// TIA Portal project "Sorting Plant Control" (V16)

(* hardware
DEVICE "S71500/ET200MP station_1"  S7-1500 station
   slot 0: "Rail_0"  Rack  6ES7 590-1***0-0AA0
   slot 0: "PM 190W 120/230VAC"  PM 190W 120/230VAC  6EP1333-4BA00
   slot 1: "Sorting Plant Controller"  CPU 1516F-3 PN/DP  6ES7 516-3FN02-0AB0  V2.8
      slot 3: "CPU display_1"  6ES7591-1BA00-0AA0
      slot 32768: "PROFINET interface_1"  X1
         slot 32769: "Port_1"  X1 P1
         slot 32770: "Port_2"  X1 P2
      slot 33024: "PROFINET interface_2"  X2
         slot 33025: "Port_1"  X2 P1
      slot 33280: "DP interface_1"  X3
      slot 34817: "Virtual CP interface port_1"  Virtual CP interface port  Virtual CP interface port
   slot 2: "DI 32x24VDC HF_1"  DI 32x24VDC HF  6ES7 521-1BL00-0AB0  V2.2
   slot 3: "DQ 32x24VDC/0.5A HF_1"  DQ 32x24VDC/0.5A HF  6ES7 522-1BL01-0AB0  V1.1
   slot 4: "AI 8xU/I/RTD/TC ST_1"  AI 8xU/I/RTD/TC ST  6ES7 531-7KF00-0AB0  V2.2
   slot 5: "AQ 4xU/I ST_1"  AQ 4xU/I ST  6ES7 532-5HD00-0AB0  V2.2
DEVICE "HMI"  TP900 Comfort
   slot 0: "HMI"  TP900 Comfort  6AV2 124-0JC01-0AX0  16.0.0.0
   slot 1: "HMI_RT_5"  TP900 Comfort  6AV2 124-0JC01-0AX0  16.0.0.0
   slot 5: "HMI._CP_1"  PROFINET Interface  16.0.0.0
      slot 1: "PROFINET Interface_1"  PROFINET Interface
         slot 1: "Port_1"  Port
         slot 2: "Port_2"  Port
   slot 7: "HMI.I/DP_CP_1"  MPI/DP Interface  16.0.0.0
*)

// ===== PLC "Sorting Plant Controller"  CPU 1516F-3 PN/DP =====

VAR_GLOBAL   // PLC tag table "Default tag table"
   "System_Byte" AT %MB1 : Byte;
   "FirstScan" AT %M1.0 : Bool;
   "DiagStatusUpdate" AT %M1.1 : Bool;
   "AlwaysTRUE" AT %M1.2 : Bool;
   "AlwaysFALSE" AT %M1.3 : Bool;
   "Clock_Byte" AT %MB0 : Byte;
   "Clock_10Hz" AT %M0.0 : Bool;
   "Clock_5Hz" AT %M0.1 : Bool;
   "Clock_2.5Hz" AT %M0.2 : Bool;
   "Clock_2Hz" AT %M0.3 : Bool;
   "Clock_1.25Hz" AT %M0.4 : Bool;
   "Clock_1Hz" AT %M0.5 : Bool;
   "Clock_0.625Hz" AT %M0.6 : Bool;
   "Clock_0.5Hz" AT %M0.7 : Bool;
   "Tag_1" AT %M2.0 : Bool;
   "Tag_2" AT %M2.1 : Bool;
   "Tag_3" AT %M2.2 : Bool;
   "Tag_4" AT %M2.3 : Bool;
   "Tag_5" AT %M2.4 : Bool;
   "Tag_6" AT %M2.5 : Bool;
   "Tag_7" AT %M2.6 : Bool;
   "Tag_8" AT %M2.7 : Bool;
END_VAR

VAR_GLOBAL   // PLC tag table "Sorting Plant Tags"
   "csLightSensorCube_Detected" AT %I0.0 : Bool;   // 0: cube workpiece not detected; 1: cube workpiece detected by the light sensor
   "csLightSensorCylinder_Detected" AT %I0.1 : Bool;   // 0: cylinder workpiece not detected; 1: cylinder workpiece detected by the light sensor
   "csLightSensorWorkpiece_Detected" AT %I0.2 : Bool;   // 0: light sensor did not detect a workpiece, 1: light sensor detected a workpiece
   "csLimitSwitchCylinderNotExtended_Activated" AT %I0.3 : Bool;   // 0: the cylinder is fully extended; 1: the cylinder is not fully extended
   "csLimitSwitchCylinderRetracted_Activated" AT %I0.4 : Bool;   // 0: the cylinder is not fully retracted; 1: the cylinder is fully retracted
   "osWorkpieceCylinder_SetActive" AT %Q0.0 : Bool;   // 0: cylinder workpiece are not produced; 1: cylinder workpiece are produced
   "osWorkpieceCube_SetActive" AT %Q0.1 : Bool;   // 0: cube workpiece are not produced; 1: cube workpiece are produced
   "pcCylinderHeadRetract_SetActive" AT %Q0.2 : Bool;   // 0: do not retract push cylinder; 1: retract push cylinder
   "pcCylinderHeadExtend_SetActive" AT %Q0.3 : Bool;   // 0: do not extend push cylinder; 1: extend push cylinder
   "scConveyorLongConstSpeed_SetActive" AT %Q0.4 : Bool;   // 0: do not move the long conveyor at constant speed; 1: move the long conveyor at constant speed
   "scConveyorLongVarSpeed_SetActive" AT %Q0.5 : Bool;   // 0: do not move the long conveyor at variable speed; 1: move the long conveyor at variable speed
   "scConveyorShortConstSpeed_SetActive" AT %Q0.6 : Bool;   // 0: do not move the short conveyor at constant speed; 1: move the short conveyor at constant speed
   "scConveyorShortVarSpeed_SetActive" AT %Q0.7 : Bool;   // 0: do not move the short conveyor at variable speed; 1: move the short conveyor at variable speed
   "scConveyorLongVarSpeed_SetSpeed" AT %QD64 : Real;   // variable velocity for long conveyor belt in m/s
   "scConveyorShortVarSpeed_SetSpeed" AT %QD68 : Real;   // variable velocity for short conveyor belt in m/s
END_VAR

DATA_BLOCK "Control_HMI"   // DB1
{ S7_Optimized_Access := 'TRUE' }
VERSION : 0.1
   VAR RETAIN
      toHMI : Struct
         resetStatus : Bool;
         numWorkpieces : USInt;
         numCylinders : USInt;
         numCubes : USInt;
         Error : Bool;
         ErrorID : Word;
      END_STRUCT;
      fromHMI : Struct
         resetSimulation : Bool;
         generateWorkpieces : Bool;
         cylinderCommand : Struct
            extendCylinder : Bool;
            retractCylinder : Bool;
         END_STRUCT;
         shortConveyor : Struct
            constSpeedControl : Bool;
            varSpeedControl : Bool;
            varSpeedPercentage : Real;   // % value
         END_STRUCT;
         longConveyor : Struct
            constSpeedControl : Bool;
            varSpeedControl : Bool;
            varSpeedPercentage : Real;   // % value
         END_STRUCT;
      END_STRUCT;
   END_VAR
BEGIN
END_DATA_BLOCK

DATA_BLOCK "SortingPlantControl_DB"   // DB2
{ S7_Optimized_Access := 'TRUE' }
VERSION : 0.1
// stored: InstanceOfName SortingPlantControl
"SortingPlantControl"
BEGIN
END_DATA_BLOCK

FUNCTION_BLOCK "SortingPlantControl"   // FB1, LAD
{ S7_Optimized_Access := 'TRUE' }
VERSION : 0.1
   VAR_INPUT
      "Light Sensor Cube" : Bool;
      "Light Sensor Cylinder" : Bool;
      "Light Sensor Workpiece" : Bool;
      "Limit Switch Cylinder NotExtended" : Bool;
      "Limit Switch Cylinder Retracted" : Bool;
      "Cylinder Extend Command" : Bool;
      "Cylinder Retract Command" : Bool;
      "Long Conveyor Constant Speed Command" : Bool;
      "Long Conveyor Var Speed Command" : Bool;
      "Long Conveyor Var Speed Percentage" : Real;
      "Short Conveyor Constant Speed Command" : Bool;
      "Short Conveyor Var Speed Command" : Bool;
      "Short Conveyor Var Speed Percentage" : Real;
      "Generate Workpieces" : Bool;
      "Total Workpiece Counter Value" : USInt;
      "Cylinder Counter Value" : USInt;
      "Cube Counter Value" : USInt;
   END_VAR
   VAR_OUTPUT
      Error : Bool;
      ErrorID : Word;
      "Workpiece Cylinder Generation" : Bool;
      "Workpiece Cube Generation" : Bool;
      "Cylinder Retract" : Bool;
      "Cylinder Extend" : Bool;
      "Conveyor Long Const Speed" : Bool;
      "Conveyor Long Var Speed" : Bool;
      "Conveyor Long Var Speed Setpoint" : Real;
      "Conveyor Short Const Speed" : Bool;
      "Conveyor Short Var Speed" : Bool;
      "Conveyor Long Short Speed Setpoint" : Real;
      "Total Workpiece Count Set" : USInt;
      "Cylinder Count Set" : USInt;
      "Cube Count Set" : USInt;
   END_VAR
   VAR
      CylinderControl_Instance : "CylinderControl";
      ShortConveyorControl_Instance : "ConveyorControl";
      LongConveyorControl_Instance : "ConveyorControl";
      upCounter_Workpiece : CTU_USINT;
      lightSensorWorkpieceFALLEdge : Bool;
      lightSensorCubeFALLEdge : Bool;
      upCounter_Cube : CTU_USINT;
      lightSensorCylinderFALLEdge : Bool;
      upCounter_Cylinder : CTU_USINT;
      waitTime : Time;   // in ms
      startWaitTimer : Bool;
      onTimer_Waitfunction : TON_TIME;
      cylinderInterlock : Bool;
      shortConvInterlock : Bool;
      longConvInterlock : Bool;
   END_VAR
   VAR_TEMP
      shortConvFault : Bool;
      longConvFault : Bool;
      cylFault : Bool;
      waitTimeCalc : UDInt;
      performEject : Bool;
   END_VAR
   VAR CONSTANT
      constantMaxSpeed : Real := 0.05;   // max speed in m/s for constant speed mode
      varMaxSpeed : Real := 0.15;   // max speed in m/s for variable speed mode
      optimumEjectDistance : Real := 0.02;   // optimal distance for ejection in m. In this case 20 mm
   END_VAR
   VAR_TEMP   // added for the SCL form of the ladder/FBD networks
      _w1 : Bool;
      _w2 : Bool;
      _w3 : Bool;
   END_VAR
BEGIN

REGION Network 1: Generate workpieces when triggered from HMI
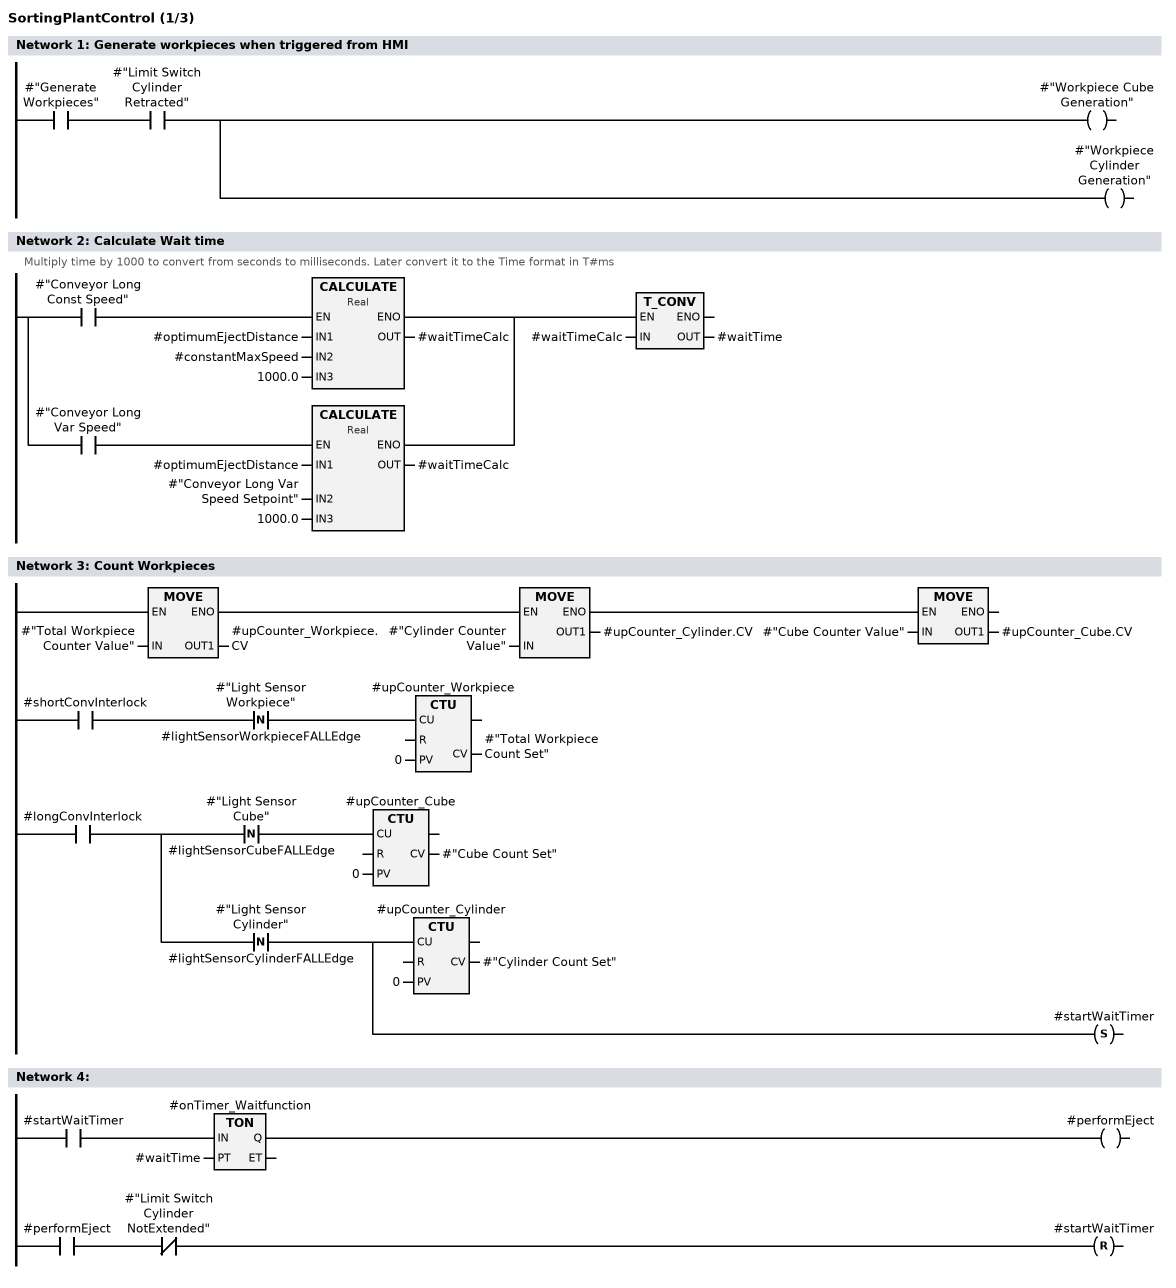
   RUNG wire#powerrail
      Contact( #"Generate Workpieces" )
      Contact( #"Limit Switch Cylinder Retracted" )
      wire#w1
      Coil( #"Workpiece Cube Generation" )
   END_RUNG
   RUNG wire#w1
      Coil( #"Workpiece Cylinder Generation" )
   END_RUNG
   // the same network as SCL:
   #"Workpiece Cube Generation" := #"Generate Workpieces" AND #"Limit Switch Cylinder Retracted";
   #"Workpiece Cylinder Generation" := #"Workpiece Cube Generation";
END_REGION

REGION Network 2: Calculate Wait time
   // Multiply time by 1000 to convert from seconds to milliseconds. Later convert it to the Time format in T#ms
   IF #"Conveyor Long Const Speed" THEN
       #waitTimeCalc := (#optimumEjectDistance / #constantMaxSpeed) * 1000.0;
   END_IF;
   IF #"Conveyor Long Var Speed" THEN
       #waitTimeCalc := (#optimumEjectDistance / #"Conveyor Long Var Speed Setpoint") * 1000.0;
   END_IF;
   IF #"Conveyor Long Const Speed" OR #"Conveyor Long Var Speed" THEN
       #waitTime := T_CONV(IN := #waitTimeCalc);
   END_IF;
END_REGION

REGION Network 3: Count Workpieces
   #upCounter_Workpiece.CV := #"Total Workpiece Counter Value";
   #upCounter_Cylinder.CV := #"Cylinder Counter Value";
   #upCounter_Cube.CV := #"Cube Counter Value";
   #_w1 := #shortConvInterlock AND NOT #"Light Sensor Workpiece" AND #lightSensorWorkpieceFALLEdge;   // falling edge of #"Light Sensor Workpiece"
   #lightSensorWorkpieceFALLEdge := #"Light Sensor Workpiece";
   #upCounter_Workpiece(CU := #_w1, PV := 0, CV => #"Total Workpiece Count Set");   // CTU
   #_w2 := #longConvInterlock AND NOT #"Light Sensor Cube" AND #lightSensorCubeFALLEdge;   // falling edge of #"Light Sensor Cube"
   #lightSensorCubeFALLEdge := #"Light Sensor Cube";
   #upCounter_Cube(CU := #_w2, PV := 0, CV => #"Cube Count Set");   // CTU
   #_w3 := #longConvInterlock AND NOT #"Light Sensor Cylinder" AND #lightSensorCylinderFALLEdge;   // falling edge of #"Light Sensor Cylinder"
   #lightSensorCylinderFALLEdge := #"Light Sensor Cylinder";
   #upCounter_Cylinder(CU := #_w3, PV := 0, CV => #"Cylinder Count Set");   // CTU
   IF #_w3 THEN #startWaitTimer := TRUE; END_IF;
END_REGION

REGION Network 4
   #onTimer_Waitfunction(IN := #startWaitTimer, PT := #waitTime);   // TON
   #performEject := #onTimer_Waitfunction.Q;
   IF #performEject AND NOT #"Limit Switch Cylinder NotExtended" THEN #startWaitTimer := FALSE; END_IF;
END_REGION

REGION Network 5: Control Pneumatic Cylinder
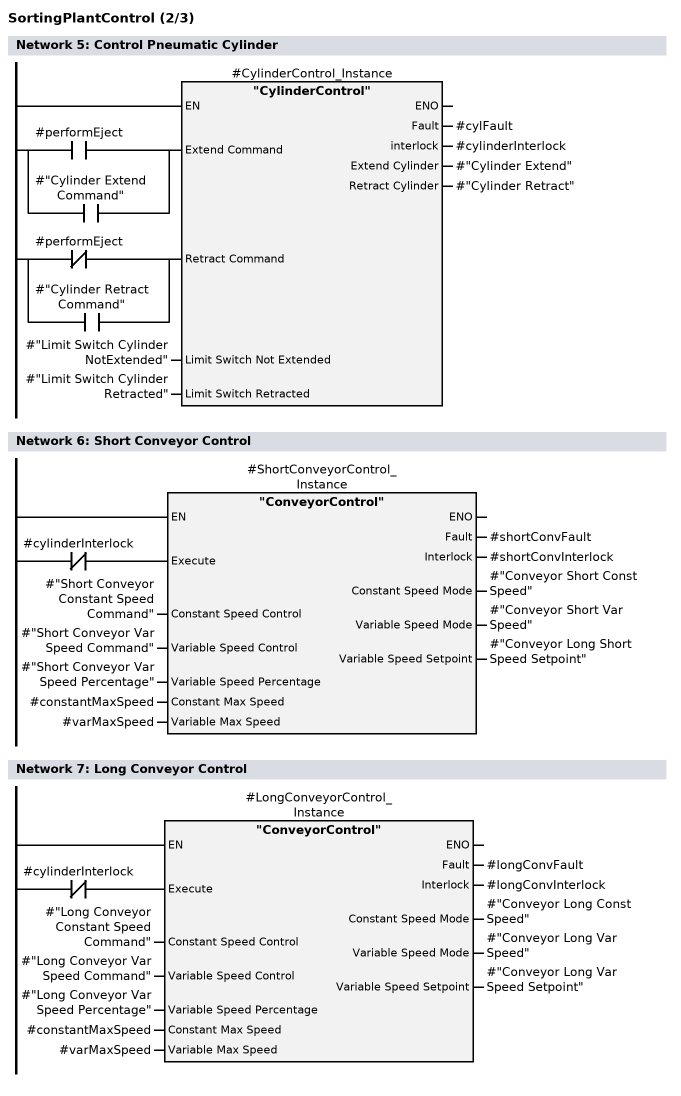
   RUNG wire#powerrail
      #CylinderControl_Instance("Extend Command" := wire#w1, "Retract Command" := wire#w2, "Limit Switch Not Extended" := #"Limit Switch Cylinder NotExtended", "Limit Switch Retracted" := #"Limit Switch Cylinder Retracted", Fault => #cylFault, interlock => #cylinderInterlock, "Extend Cylinder" => #"Cylinder Extend", "Retract Cylinder" => #"Cylinder Retract")
   END_RUNG
   RUNG wire#powerrail
      Contact( #performEject )
   END_RUNG wire#w1
   RUNG wire#powerrail
      Contact( #"Cylinder Extend Command" )
   END_RUNG wire#w1
   RUNG wire#powerrail
      I_Contact( #performEject )
   END_RUNG wire#w2
   RUNG wire#powerrail
      Contact( #"Cylinder Retract Command" )
   END_RUNG wire#w2
   // the same network as SCL:
   #CylinderControl_Instance("Extend Command" := #performEject OR #"Cylinder Extend Command",   // "CylinderControl"
                           "Retract Command" := NOT #performEject OR #"Cylinder Retract Command",
                           "Limit Switch Not Extended" := #"Limit Switch Cylinder NotExtended",
                           "Limit Switch Retracted" := #"Limit Switch Cylinder Retracted",
                           Fault => #cylFault,
                           interlock => #cylinderInterlock,
                           "Extend Cylinder" => #"Cylinder Extend",
                           "Retract Cylinder" => #"Cylinder Retract");
END_REGION

REGION Network 6: Short Conveyor Control
   RUNG wire#powerrail
      #ShortConveyorControl_Instance(Execute := wire#w1, "Constant Speed Control" := #"Short Conveyor Constant Speed Command", "Variable Speed Control" := #"Short Conveyor Var Speed Command", "Variable Speed Percentage" := #"Short Conveyor Var Speed Percentage", "Constant Max Speed" := #constantMaxSpeed, "Variable Max Speed" := #varMaxSpeed, Fault => #shortConvFault, Interlock => #shortConvInterlock, "Constant Speed Mode" => #"Conveyor Short Const Speed", "Variable Speed Mode" => #"Conveyor Short Var Speed", "Variable Speed Setpoint" => #"Conveyor Long Short Speed Setpoint")
   END_RUNG
   RUNG wire#powerrail
      I_Contact( #cylinderInterlock )
   END_RUNG wire#w1
   // the same network as SCL:
   #ShortConveyorControl_Instance(Execute := NOT #cylinderInterlock,   // "ConveyorControl"
                           "Constant Speed Control" := #"Short Conveyor Constant Speed Command",
                           "Variable Speed Control" := #"Short Conveyor Var Speed Command",
                           "Variable Speed Percentage" := #"Short Conveyor Var Speed Percentage",
                           "Constant Max Speed" := #constantMaxSpeed,
                           "Variable Max Speed" := #varMaxSpeed,
                           Fault => #shortConvFault,
                           Interlock => #shortConvInterlock,
                           "Constant Speed Mode" => #"Conveyor Short Const Speed",
                           "Variable Speed Mode" => #"Conveyor Short Var Speed",
                           "Variable Speed Setpoint" => #"Conveyor Long Short Speed Setpoint");
END_REGION

REGION Network 7: Long Conveyor Control
   RUNG wire#powerrail
      #LongConveyorControl_Instance(Execute := wire#w1, "Constant Speed Control" := #"Long Conveyor Constant Speed Command", "Variable Speed Control" := #"Long Conveyor Var Speed Command", "Variable Speed Percentage" := #"Long Conveyor Var Speed Percentage", "Constant Max Speed" := #constantMaxSpeed, "Variable Max Speed" := #varMaxSpeed, Fault => #longConvFault, Interlock => #longConvInterlock, "Constant Speed Mode" => #"Conveyor Long Const Speed", "Variable Speed Mode" => #"Conveyor Long Var Speed", "Variable Speed Setpoint" => #"Conveyor Long Var Speed Setpoint")
   END_RUNG
   RUNG wire#powerrail
      I_Contact( #cylinderInterlock )
   END_RUNG wire#w1
   // the same network as SCL:
   #LongConveyorControl_Instance(Execute := NOT #cylinderInterlock,   // "ConveyorControl"
                           "Constant Speed Control" := #"Long Conveyor Constant Speed Command",
                           "Variable Speed Control" := #"Long Conveyor Var Speed Command",
                           "Variable Speed Percentage" := #"Long Conveyor Var Speed Percentage",
                           "Constant Max Speed" := #constantMaxSpeed,
                           "Variable Max Speed" := #varMaxSpeed,
                           Fault => #longConvFault,
                           Interlock => #longConvInterlock,
                           "Constant Speed Mode" => #"Conveyor Long Const Speed",
                           "Variable Speed Mode" => #"Conveyor Long Var Speed",
                           "Variable Speed Setpoint" => #"Conveyor Long Var Speed Setpoint");
END_REGION

REGION Network 8: Trigger Fault
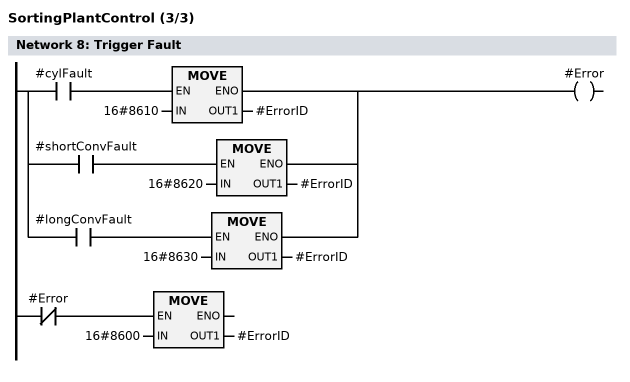
   RUNG wire#powerrail
      Contact( #cylFault )
      Move(in := 16#8610, out1 => #ErrorID)
      wire#w1
      Coil( #Error )
   END_RUNG
   RUNG wire#powerrail
      Contact( #shortConvFault )
      Move(in := 16#8620, out1 => #ErrorID)
   END_RUNG wire#w1
   RUNG wire#powerrail
      Contact( #longConvFault )
      Move(in := 16#8630, out1 => #ErrorID)
   END_RUNG wire#w1
   RUNG wire#powerrail
      I_Contact( #Error )
      Move(in := 16#8600, out1 => #ErrorID)
   END_RUNG
   // the same network as SCL:
   IF #cylFault THEN #ErrorID := 16#8610; END_IF;
   IF #shortConvFault THEN #ErrorID := 16#8620; END_IF;
   IF #longConvFault THEN #ErrorID := 16#8630; END_IF;
   #Error := #cylFault OR #shortConvFault OR #longConvFault;
   IF NOT #Error THEN #ErrorID := 16#8600; END_IF;
END_REGION
END_FUNCTION_BLOCK

FUNCTION_BLOCK "CylinderControl"   // FB2, LAD
{ S7_Optimized_Access := 'TRUE' }
VERSION : 0.1
   VAR_INPUT
      "Extend Command" : Bool;
      "Retract Command" : Bool;
      "Limit Switch Not Extended" : Bool;
      "Limit Switch Retracted" : Bool;
   END_VAR
   VAR_OUTPUT
      Fault : Bool;
      interlock : Bool;
      "Extend Cylinder" : Bool;
      "Retract Cylinder" : Bool;
   END_VAR
BEGIN

REGION Network 1: Trigger fault when the cylinder is set to extend and retract at the same time
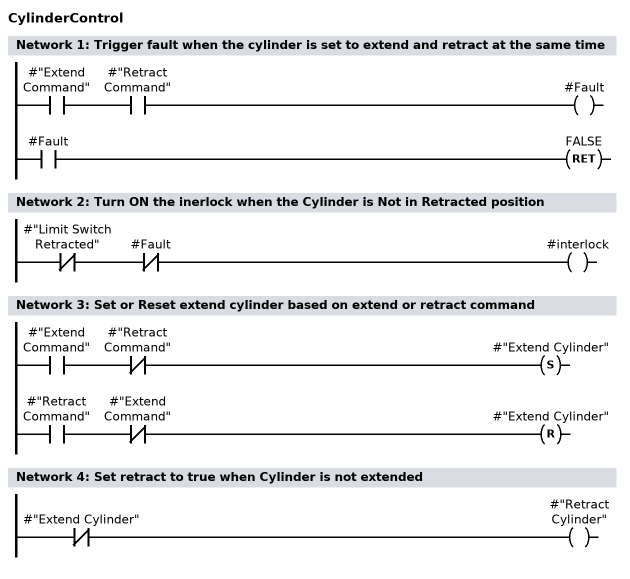
   #Fault := #"Extend Command" AND #"Retract Command";
   IF #Fault THEN
       ENO := FALSE;
       RETURN;
   END_IF;
END_REGION

REGION Network 2: Turn ON the inerlock when the Cylinder is Not in Retracted position
   RUNG wire#powerrail
      I_Contact( #"Limit Switch Retracted" )
      I_Contact( #Fault )
      Coil( #interlock )
   END_RUNG
   // the same network as SCL:
   #interlock := NOT #"Limit Switch Retracted" AND NOT #Fault;
END_REGION

REGION Network 3: Set or Reset extend cylinder based on extend or retract command
   RUNG wire#powerrail
      Contact( #"Extend Command" )
      I_Contact( #"Retract Command" )
      S_Coil( #"Extend Cylinder" )
   END_RUNG
   RUNG wire#powerrail
      Contact( #"Retract Command" )
      I_Contact( #"Extend Command" )
      R_Coil( #"Extend Cylinder" )
   END_RUNG
   // the same network as SCL:
   IF #"Extend Command" AND NOT #"Retract Command" THEN #"Extend Cylinder" := TRUE; END_IF;
   IF #"Retract Command" AND NOT #"Extend Command" THEN #"Extend Cylinder" := FALSE; END_IF;
END_REGION

REGION Network 4: Set retract to true when Cylinder is not extended
   RUNG wire#powerrail
      I_Contact( #"Extend Cylinder" )
      Coil( #"Retract Cylinder" )
   END_RUNG
   // the same network as SCL:
   #"Retract Cylinder" := NOT #"Extend Cylinder";
END_REGION
END_FUNCTION_BLOCK

FUNCTION_BLOCK "ConveyorControl"   // FB3, LAD
{ S7_Optimized_Access := 'TRUE' }
VERSION : 0.1
   VAR_INPUT
      Execute : Bool;
      "Constant Speed Control" : Bool;
      "Variable Speed Control" : Bool;
      "Variable Speed Percentage" : Real;
      "Constant Max Speed" : Real;
      "Variable Max Speed" : Real;
   END_VAR
   VAR_OUTPUT
      Fault : Bool;
      Interlock : Bool;
      "Constant Speed Mode" : Bool;
      "Variable Speed Mode" : Bool;
      "Variable Speed Setpoint" : Real;
   END_VAR
   VAR_TEMP
      varSpeedSetpoint : Real;
   END_VAR
BEGIN

REGION Network 1: Fault
   // Trigger a fault if the conveyor is controlled both by constant and variable mode
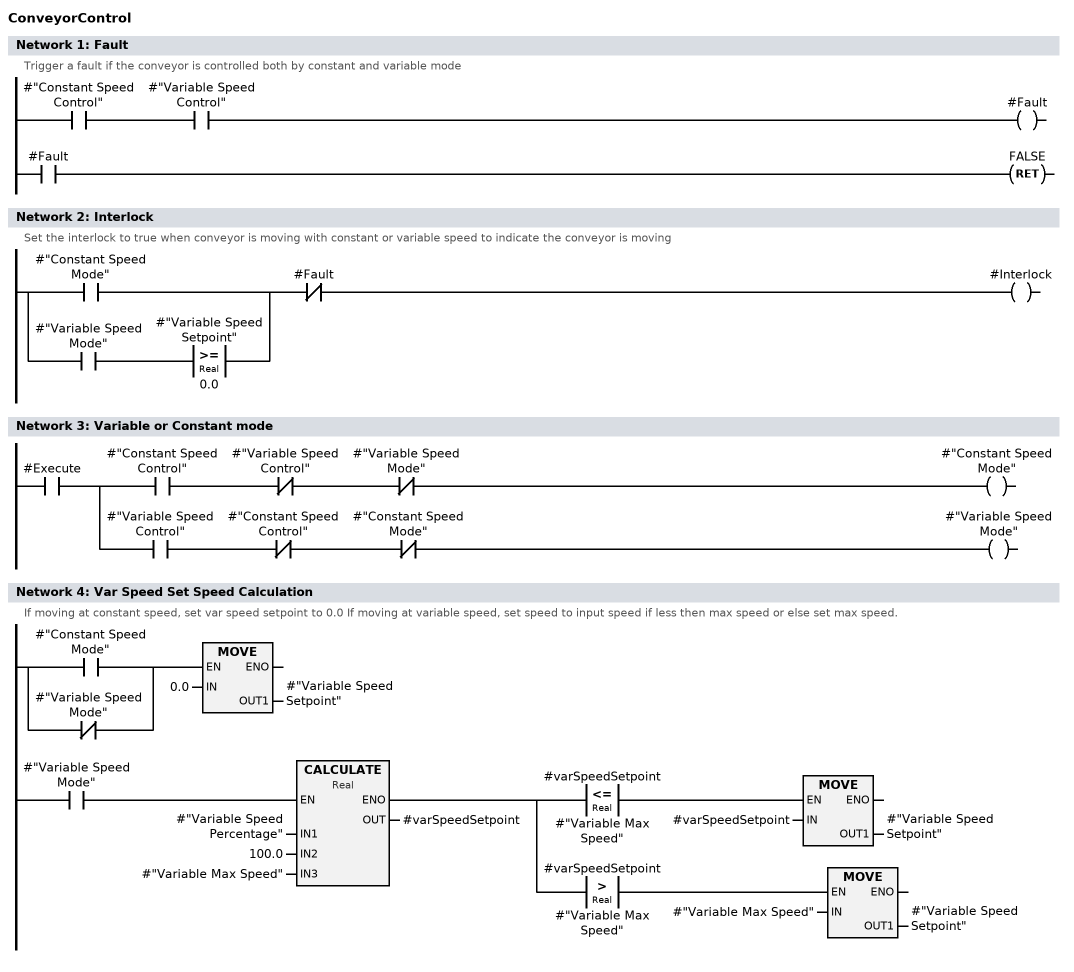
   #Fault := #"Constant Speed Control" AND #"Variable Speed Control";
   IF #Fault THEN
       ENO := FALSE;
       RETURN;
   END_IF;
END_REGION

REGION Network 2: Interlock
   // Set the interlock to true when conveyor is moving with constant or variable speed to indicate the conveyor is moving
   RUNG wire#powerrail
      Contact( #"Constant Speed Mode" )
      wire#w1
      I_Contact( #Fault )
      Coil( #Interlock )
   END_RUNG
   RUNG wire#powerrail
      Contact( #"Variable Speed Mode" )
      { S7_Templates := "SrcType := Real" } GE_Contact(in1 := #"Variable Speed Setpoint", in2 := 0.0)
   END_RUNG wire#w1
   // the same network as SCL:
   #Interlock := (#"Constant Speed Mode" OR (#"Variable Speed Mode" AND (#"Variable Speed Setpoint" >= 0.0))) AND NOT #Fault;
END_REGION

REGION Network 3: Variable or Constant mode
   RUNG wire#powerrail
      Contact( #Execute )
      wire#w1
      Contact( #"Constant Speed Control" )
      I_Contact( #"Variable Speed Control" )
      I_Contact( #"Variable Speed Mode" )
      Coil( #"Constant Speed Mode" )
   END_RUNG
   RUNG wire#w1
      Contact( #"Variable Speed Control" )
      I_Contact( #"Constant Speed Control" )
      I_Contact( #"Constant Speed Mode" )
      Coil( #"Variable Speed Mode" )
   END_RUNG
   // the same network as SCL:
   #"Constant Speed Mode" := #Execute AND #"Constant Speed Control" AND NOT #"Variable Speed Control" AND NOT #"Variable Speed Mode";
   #"Variable Speed Mode" := #Execute AND #"Variable Speed Control" AND NOT #"Constant Speed Control" AND NOT #"Constant Speed Mode";
END_REGION

REGION Network 4: Var Speed Set Speed Calculation
   // If moving at constant speed, set var speed setpoint to 0.0 If moving at variable speed, set speed to input speed if less then max speed or else set max speed.
   RUNG wire#powerrail
      Contact( #"Constant Speed Mode" )
      wire#w1
      Move(in := 0.0, out1 => #"Variable Speed Setpoint")
   END_RUNG
   RUNG wire#powerrail
      I_Contact( #"Variable Speed Mode" )
   END_RUNG wire#w1
   RUNG wire#powerrail
      Contact( #"Variable Speed Mode" )
      { S7_Templates := "SrcType := Real"; S7_Expression := "(IN1 / IN2) * IN3" } Calculate(in1 := #"Variable Speed Percentage", in2 := 100.0, in3 := #"Variable Max Speed", out => #varSpeedSetpoint)
      wire#w2
      { S7_Templates := "SrcType := Real" } LE_Contact(in1 := #varSpeedSetpoint, in2 := #"Variable Max Speed")
      Move(in := #varSpeedSetpoint, out1 => #"Variable Speed Setpoint")
   END_RUNG
   RUNG wire#w2
      { S7_Templates := "SrcType := Real" } GT_Contact(in1 := #varSpeedSetpoint, in2 := #"Variable Max Speed")
      Move(in := #"Variable Max Speed", out1 => #"Variable Speed Setpoint")
   END_RUNG
   // the same network as SCL:
   IF #"Constant Speed Mode" OR NOT #"Variable Speed Mode" THEN #"Variable Speed Setpoint" := 0.0; END_IF;
   IF #"Variable Speed Mode" THEN
       #varSpeedSetpoint := (#"Variable Speed Percentage" / 100.0) * #"Variable Max Speed";
   END_IF;
   IF #"Variable Speed Mode" AND (#varSpeedSetpoint <= #"Variable Max Speed") THEN
       #"Variable Speed Setpoint" := #varSpeedSetpoint;
   END_IF;
   IF #"Variable Speed Mode" AND (#varSpeedSetpoint > #"Variable Max Speed") THEN
       #"Variable Speed Setpoint" := #"Variable Max Speed";
   END_IF;
END_REGION
END_FUNCTION_BLOCK

FUNCTION "ResetSimulation" : Void   // FC1, LAD
{ S7_Optimized_Access := 'TRUE' }
VERSION : 0.1
   VAR_OUTPUT
      osWorkpieceCube_SetActive : Bool;
      osWorkpieceCylinder_SetActive : Bool;
      pcCylinderHeadRetract_SetActive : Bool;
      pcCylinderHeadExtend_SetActive : Bool;
      scConveyorLongConstSpeed_SetActive : Bool;
      scConveyorLongVarSpeed_SetActive : Bool;
      scConveyorShortConstSpeed_SetActive : Bool;
      scConveyorShortVarSpeed_SetActive : Bool;
      scConveyorLongVarSpeed_SetSpeed : Real;
      scConveyorShortVarSpeed_SetSpeed : Real;
      "Workpiece Counter" : USInt;
      "Cylindrical Counter" : USInt;
      "Cube Counter" : USInt;
   END_VAR
BEGIN

REGION Network 1: Reset PLC Tags and Counter
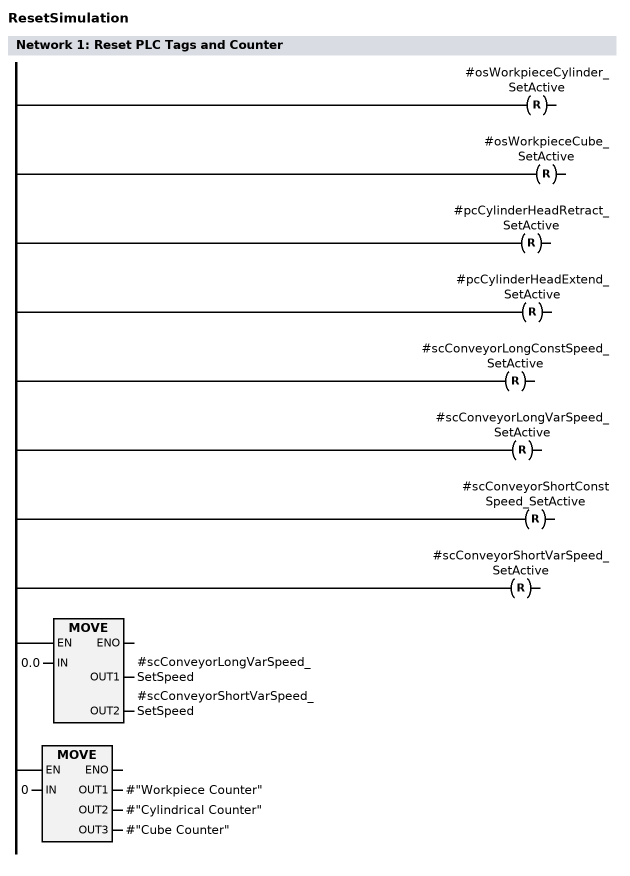
   RUNG wire#powerrail
      R_Coil( #osWorkpieceCylinder_SetActive )
   END_RUNG
   RUNG wire#powerrail
      R_Coil( #osWorkpieceCube_SetActive )
   END_RUNG
   RUNG wire#powerrail
      R_Coil( #pcCylinderHeadRetract_SetActive )
   END_RUNG
   RUNG wire#powerrail
      R_Coil( #pcCylinderHeadExtend_SetActive )
   END_RUNG
   RUNG wire#powerrail
      R_Coil( #scConveyorLongConstSpeed_SetActive )
   END_RUNG
   RUNG wire#powerrail
      R_Coil( #scConveyorLongVarSpeed_SetActive )
   END_RUNG
   RUNG wire#powerrail
      R_Coil( #scConveyorShortConstSpeed_SetActive )
   END_RUNG
   RUNG wire#powerrail
      R_Coil( #scConveyorShortVarSpeed_SetActive )
   END_RUNG
   RUNG wire#powerrail
      Move(in := 0.0, out1 => #scConveyorLongVarSpeed_SetSpeed, out2 => #scConveyorShortVarSpeed_SetSpeed)
   END_RUNG
   RUNG wire#powerrail
      Move(in := 0, out1 => #"Workpiece Counter", out2 => #"Cylindrical Counter", out3 => #"Cube Counter")
   END_RUNG
   // the same network as SCL:
   #osWorkpieceCylinder_SetActive := FALSE;
   #osWorkpieceCube_SetActive := FALSE;
   #pcCylinderHeadRetract_SetActive := FALSE;
   #pcCylinderHeadExtend_SetActive := FALSE;
   #scConveyorLongConstSpeed_SetActive := FALSE;
   #scConveyorLongVarSpeed_SetActive := FALSE;
   #scConveyorShortConstSpeed_SetActive := FALSE;
   #scConveyorShortVarSpeed_SetActive := FALSE;
   #scConveyorLongVarSpeed_SetSpeed := 0.0;
   #scConveyorShortVarSpeed_SetSpeed := 0.0;
   #"Workpiece Counter" := 0;
   #"Cylindrical Counter" := 0;
   #"Cube Counter" := 0;
END_REGION
END_FUNCTION

ORGANIZATION_BLOCK "Main"   // OB1, LAD, ProgramCycle
TITLE = "Main Program Sweep (Cycle)"
{ S7_Optimized_Access := 'TRUE' }
VERSION : 0.1
   VAR_INPUT
      Initial_Call : Bool;   // Initial call of this OB
      Remanence : Bool;   // =True, if remanent data are available
   END_VAR
   VAR_TEMP   // added for the SCL form of the ladder/FBD networks
      _w1 : Bool;
   END_VAR
BEGIN

REGION Network 1: Reset the Simulation and PLC Tags
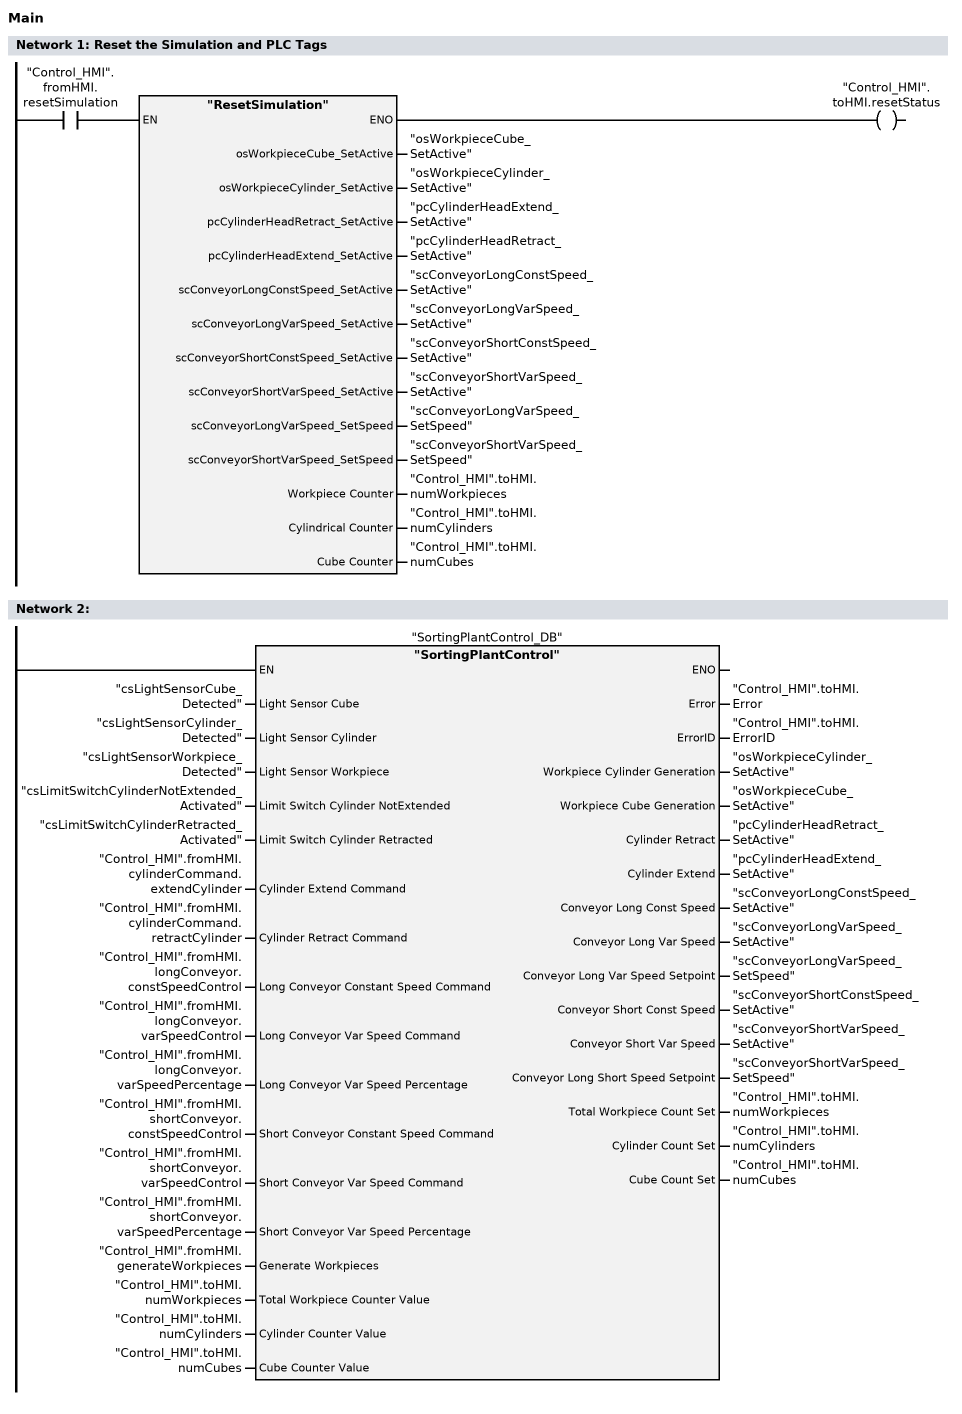
   RUNG wire#powerrail
      Contact( "Control_HMI".fromHMI.resetSimulation )
      "ResetSimulation"(osWorkpieceCube_SetActive => "osWorkpieceCube_SetActive", osWorkpieceCylinder_SetActive => "osWorkpieceCylinder_SetActive", pcCylinderHeadRetract_SetActive => "pcCylinderHeadExtend_SetActive", pcCylinderHeadExtend_SetActive => "pcCylinderHeadRetract_SetActive", scConveyorLongConstSpeed_SetActive => "scConveyorLongConstSpeed_SetActive", scConveyorLongVarSpeed_SetActive => "scConveyorLongVarSpeed_SetActive", scConveyorShortConstSpeed_SetActive => "scConveyorShortConstSpeed_SetActive", scConveyorShortVarSpeed_SetActive => "scConveyorShortVarSpeed_SetActive", scConveyorLongVarSpeed_SetSpeed => "scConveyorLongVarSpeed_SetSpeed", scConveyorShortVarSpeed_SetSpeed => "scConveyorShortVarSpeed_SetSpeed", "Workpiece Counter" => "Control_HMI".toHMI.numWorkpieces, "Cylindrical Counter" => "Control_HMI".toHMI.numCylinders, "Cube Counter" => "Control_HMI".toHMI.numCubes)
      Coil( "Control_HMI".toHMI.resetStatus )
   END_RUNG
   // the same network as SCL:
   "ResetSimulation"(EN := "Control_HMI".fromHMI.resetSimulation,
                     osWorkpieceCube_SetActive => "osWorkpieceCube_SetActive",
                     osWorkpieceCylinder_SetActive => "osWorkpieceCylinder_SetActive",
                     pcCylinderHeadRetract_SetActive => "pcCylinderHeadExtend_SetActive",
                     pcCylinderHeadExtend_SetActive => "pcCylinderHeadRetract_SetActive",
                     scConveyorLongConstSpeed_SetActive => "scConveyorLongConstSpeed_SetActive",
                     scConveyorLongVarSpeed_SetActive => "scConveyorLongVarSpeed_SetActive",
                     scConveyorShortConstSpeed_SetActive => "scConveyorShortConstSpeed_SetActive",
                     scConveyorShortVarSpeed_SetActive => "scConveyorShortVarSpeed_SetActive",
                     scConveyorLongVarSpeed_SetSpeed => "scConveyorLongVarSpeed_SetSpeed",
                     scConveyorShortVarSpeed_SetSpeed => "scConveyorShortVarSpeed_SetSpeed",
                     "Workpiece Counter" => "Control_HMI".toHMI.numWorkpieces,
                     "Cylindrical Counter" => "Control_HMI".toHMI.numCylinders,
                     "Cube Counter" => "Control_HMI".toHMI.numCubes,
                     ENO => #_w1);
   "Control_HMI".toHMI.resetStatus := #_w1;
END_REGION

REGION Network 2
   RUNG wire#powerrail
      "SortingPlantControl_DB"("Light Sensor Cube" := "csLightSensorCube_Detected", "Light Sensor Cylinder" := "csLightSensorCylinder_Detected", "Light Sensor Workpiece" := "csLightSensorWorkpiece_Detected", "Limit Switch Cylinder NotExtended" := "csLimitSwitchCylinderNotExtended_Activated", "Limit Switch Cylinder Retracted" := "csLimitSwitchCylinderRetracted_Activated", "Cylinder Extend Command" := "Control_HMI".fromHMI.cylinderCommand.extendCylinder, "Cylinder Retract Command" := "Control_HMI".fromHMI.cylinderCommand.retractCylinder, "Long Conveyor Constant Speed Command" := "Control_HMI".fromHMI.longConveyor.constSpeedControl, "Long Conveyor Var Speed Command" := "Control_HMI".fromHMI.longConveyor.varSpeedControl, "Long Conveyor Var Speed Percentage" := "Control_HMI".fromHMI.longConveyor.varSpeedPercentage, "Short Conveyor Constant Speed Command" := "Control_HMI".fromHMI.shortConveyor.constSpeedControl, "Short Conveyor Var Speed Command" := "Control_HMI".fromHMI.shortConveyor.varSpeedControl, "Short Conveyor Var Speed Percentage" := "Control_HMI".fromHMI.shortConveyor.varSpeedPercentage, "Generate Workpieces" := "Control_HMI".fromHMI.generateWorkpieces, "Total Workpiece Counter Value" := "Control_HMI".toHMI.numWorkpieces, "Cylinder Counter Value" := "Control_HMI".toHMI.numCylinders, "Cube Counter Value" := "Control_HMI".toHMI.numCubes, Error => "Control_HMI".toHMI.Error, ErrorID => "Control_HMI".toHMI.ErrorID, "Workpiece Cylinder Generation" => "osWorkpieceCylinder_SetActive", "Workpiece Cube Generation" => "osWorkpieceCube_SetActive", "Cylinder Retract" => "pcCylinderHeadRetract_SetActive", "Cylinder Extend" => "pcCylinderHeadExtend_SetActive", "Conveyor Long Const Speed" => "scConveyorLongConstSpeed_SetActive", "Conveyor Long Var Speed" => "scConveyorLongVarSpeed_SetActive", "Conveyor Long Var Speed Setpoint" => "scConveyorLongVarSpeed_SetSpeed", "Conveyor Short Const Speed" => "scConveyorShortConstSpeed_SetActive", "Conveyor Short Var Speed" => "scConveyorShortVarSpeed_SetActive", "Conveyor Long Short Speed Setpoint" => "scConveyorShortVarSpeed_SetSpeed", "Total Workpiece Count Set" => "Control_HMI".toHMI.numWorkpieces, "Cylinder Count Set" => "Control_HMI".toHMI.numCylinders, "Cube Count Set" => "Control_HMI".toHMI.numCubes)
   END_RUNG
   // the same network as SCL:
   "SortingPlantControl_DB"("Light Sensor Cube" := "csLightSensorCube_Detected",   // "SortingPlantControl"
                           "Light Sensor Cylinder" := "csLightSensorCylinder_Detected",
                           "Light Sensor Workpiece" := "csLightSensorWorkpiece_Detected",
                           "Limit Switch Cylinder NotExtended" := "csLimitSwitchCylinderNotExtended_Activated",
                           "Limit Switch Cylinder Retracted" := "csLimitSwitchCylinderRetracted_Activated",
                           "Cylinder Extend Command" := "Control_HMI".fromHMI.cylinderCommand.extendCylinder,
                           "Cylinder Retract Command" := "Control_HMI".fromHMI.cylinderCommand.retractCylinder,
                           "Long Conveyor Constant Speed Command" := "Control_HMI".fromHMI.longConveyor.constSpeedControl,
                           "Long Conveyor Var Speed Command" := "Control_HMI".fromHMI.longConveyor.varSpeedControl,
                           "Long Conveyor Var Speed Percentage" := "Control_HMI".fromHMI.longConveyor.varSpeedPercentage,
                           "Short Conveyor Constant Speed Command" := "Control_HMI".fromHMI.shortConveyor.constSpeedControl,
                           "Short Conveyor Var Speed Command" := "Control_HMI".fromHMI.shortConveyor.varSpeedControl,
                           "Short Conveyor Var Speed Percentage" := "Control_HMI".fromHMI.shortConveyor.varSpeedPercentage,
                           "Generate Workpieces" := "Control_HMI".fromHMI.generateWorkpieces,
                           "Total Workpiece Counter Value" := "Control_HMI".toHMI.numWorkpieces,
                           "Cylinder Counter Value" := "Control_HMI".toHMI.numCylinders,
                           "Cube Counter Value" := "Control_HMI".toHMI.numCubes,
                           Error => "Control_HMI".toHMI.Error,
                           ErrorID => "Control_HMI".toHMI.ErrorID,
                           "Workpiece Cylinder Generation" => "osWorkpieceCylinder_SetActive",
                           "Workpiece Cube Generation" => "osWorkpieceCube_SetActive",
                           "Cylinder Retract" => "pcCylinderHeadRetract_SetActive",
                           "Cylinder Extend" => "pcCylinderHeadExtend_SetActive",
                           "Conveyor Long Const Speed" => "scConveyorLongConstSpeed_SetActive",
                           "Conveyor Long Var Speed" => "scConveyorLongVarSpeed_SetActive",
                           "Conveyor Long Var Speed Setpoint" => "scConveyorLongVarSpeed_SetSpeed",
                           "Conveyor Short Const Speed" => "scConveyorShortConstSpeed_SetActive",
                           "Conveyor Short Var Speed" => "scConveyorShortVarSpeed_SetActive",
                           "Conveyor Long Short Speed Setpoint" => "scConveyorShortVarSpeed_SetSpeed",
                           "Total Workpiece Count Set" => "Control_HMI".toHMI.numWorkpieces,
                           "Cylinder Count Set" => "Control_HMI".toHMI.numCylinders,
                           "Cube Count Set" => "Control_HMI".toHMI.numCubes);
END_REGION
END_ORGANIZATION_BLOCK

(* ===== HMI "HMI_RT_5" =====
system functions are stored by id; their names below are inferred from use
connection "HMI_Connection_7": 
connection "HMI_Connection_1": ETHERNET, S7_1500_OMS

HMI tags "Template"
   "MainNavigationState" : Int, internal
   "SubNavigationState" : Int, internal
   "CurrentUserName" : WString[18], internal
   "DiagState" : Int, internal
   "PopUpBackground" : Bool, internal
   "UserName" : WString[20], internal
   "Password" : WString[20], internal
   "UserIsLoggedIn" : Bool, internal
   "CodeView" : Bool, internal
   "Brightness" : Int, internal
   "CurrentLanguage" : Bool, internal
   "CurrentRecipeName" : WString[30], internal
   "CurrentMachineState" : Int, internal
   "OptionPanelNavigationState" : Int, internal
   "ButtonDown" : Bool, internal
   "ThirdLevelNavigationState" : Int, internal
   "StartScreenName" : WString[60], internal
   "InScreenTabState" : Int, internal
   "DummyTagBool" : Bool, internal
   "DummyTagInt1" : Int, internal
   "DummyTagInt2" : Int, internal
   "DummyTagInt3" : Int, internal
   "DummyDeltaReal" : LReal, internal
   "DummTagReal1" : LReal, internal
   "DummyDeltaInt" : Int, internal

HMI tags "PLC_DB"
   "Control_HMI_toHMI_resetStatus" : Bool = PLC Control_HMI.toHMI.resetStatus, 100 ms
   "Control_HMI_toHMI_numWorkpieces" : USInt = PLC Control_HMI.toHMI.numWorkpieces, 100 ms
   "Control_HMI_toHMI_numCylinders" : USInt = PLC Control_HMI.toHMI.numCylinders, 100 ms
   "Control_HMI_toHMI_numCubes" : USInt = PLC Control_HMI.toHMI.numCubes, 100 ms
   "Control_HMI_toHMI_Error" : Bool = PLC Control_HMI.toHMI.Error, 100 ms
   "Control_HMI_toHMI_ErrorID" : Word = PLC Control_HMI.toHMI.ErrorID, 100 ms
   "Control_HMI_fromHMI_resetSimulation" : Bool = PLC Control_HMI.fromHMI.resetSimulation, 100 ms
   "Control_HMI_fromHMI_generateWorkpieces" : Bool = PLC Control_HMI.fromHMI.generateWorkpieces, 100 ms
   "Control_HMI_fromHMI_cylinderCommand_extendCylinder" : Bool = PLC Control_HMI.fromHMI.cylinderCommand.extendCylinder, 100 ms
   "Control_HMI_fromHMI_cylinderCommand_retractCylinder" : Bool = PLC Control_HMI.fromHMI.cylinderCommand.retractCylinder, 100 ms
   "Control_HMI_fromHMI_shortConveyor_constSpeedControl" : Bool = PLC Control_HMI.fromHMI.shortConveyor.constSpeedControl, 100 ms
   "Control_HMI_fromHMI_shortConveyor_varSpeedControl" : Bool = PLC Control_HMI.fromHMI.shortConveyor.varSpeedControl, 100 ms
   "Control_HMI_fromHMI_shortConveyor_varSpeedPercentage" : Real = PLC Control_HMI.fromHMI.shortConveyor.varSpeedPercentage, 100 ms
   "Control_HMI_fromHMI_longConveyor_constSpeedControl" : Bool = PLC Control_HMI.fromHMI.longConveyor.constSpeedControl, 100 ms
   "Control_HMI_fromHMI_longConveyor_varSpeedControl" : Bool = PLC Control_HMI.fromHMI.longConveyor.varSpeedControl, 100 ms
   "Control_HMI_fromHMI_longConveyor_varSpeedPercentage" : Real = PLC Control_HMI.fromHMI.longConveyor.varSpeedPercentage, 100 ms

HMI tags "PLC_Tags"
   "csLightSensorCube_Detected" : Bool = PLC csLightSensorCube_Detected AT %I0.0, 100 ms
   "csLightSensorCylinder_Detected" : Bool = PLC csLightSensorCylinder_Detected AT %I0.1, 100 ms
   "csLightSensorWorkpiece_Detected" : Bool = PLC csLightSensorWorkpiece_Detected AT %I0.2, 100 ms
   "csLimitSwitchCylinderNotExtended_Activated" : Bool = PLC csLimitSwitchCylinderNotExtended_Activated AT %I0.3, 100 ms
   "csLimitSwitchCylinderRetracted_Activated" : Bool = PLC csLimitSwitchCylinderRetracted_Activated AT %I0.4, 100 ms
   "osWorkpieceCube_SetActive" : Bool = PLC osWorkpieceCube_SetActive AT %Q0.1, 100 ms
   "osWorkpieceCylinder_SetActive" : Bool = PLC osWorkpieceCylinder_SetActive AT %Q0.0, 100 ms
   "pcCylinderHeadExtend_SetActive" : Bool = PLC pcCylinderHeadExtend_SetActive AT %Q0.3, 100 ms
   "pcCylinderHeadRetract_SetActive" : Bool = PLC pcCylinderHeadRetract_SetActive AT %Q0.2, 100 ms
   "scConveyorLongConstSpeed_SetActive" : Bool = PLC scConveyorLongConstSpeed_SetActive AT %Q0.4, 100 ms
   "scConveyorLongVarSpeed_SetActive" : Bool = PLC scConveyorLongVarSpeed_SetActive AT %Q0.5, 100 ms
   "scConveyorLongVarSpeed_SetSpeed" : Real = PLC scConveyorLongVarSpeed_SetSpeed AT %QD64, 100 ms
   "scConveyorShortConstSpeed_SetActive" : Bool = PLC scConveyorShortConstSpeed_SetActive AT %Q0.6, 100 ms
   "scConveyorShortVarSpeed_SetActive" : Bool = PLC scConveyorShortVarSpeed_SetActive AT %Q0.7, 100 ms
   "scConveyorShortVarSpeed_SetSpeed" : Real = PLC scConveyorShortVarSpeed_SetSpeed AT %QD68, 100 ms

text list "Machine State": 0 'Undefined / Kein Job'; 1 'Production / Produktion'; 2 'Startup / Anlauf'; 3 'Paused / Pausiert'; 4 'Stopped / Gestoppt'; 5 'Shutdown / Beenden'; 6 'Undefined / UNBEKANNT'

text list "timeRange": 1 'Hours / Stunden'; 2 'Days / Tage'; 3 'Weeks / Wochen'; 4 'Months / Monate'; 5 'Years / Jahre'

text list "MachineState_Farfield": 0..1 '???'; 1 'OK'; 2 'ERROR / FEHLER'; 3 'PAUSED / HALT'

text list "Foil Types": 0..1 '120 - 1mm - Transparent'; 1 '120 - 3mm - Transparent'; 2 '240 - 1mm - Transparent'; 3 '240 - 3mm - Transparent'

text list "FunctionState": 0 'Disabled / Deaktiviert'; 1 'Enabled / Aktiviert'

text list "GroundPos": 0 'No / Nein'; 1 'Yes / Ja'

text list "State": 0 'Off / Aus'; 1 'On / An'

graphic list "DiagState": 0 'DiagOkay'; 1 'DiagWarning_1'; 2 'DiagDefault'

graphic list "DiagState_1": 0 'DiagOkay_1'; 1 'DiagWarning'; 2 'DiagDefault'

graphic list "DiagState_2": 0 'DiagOkay_1'; 1 'DiagWarning'; 2 'DiagDefault'

graphic list "DiagState_3": 0 'DiagOkay_White'; 1 'DiagWarning_White'; 2 'Circle'

graphic list "State": 0..1 'OK'; 3 'Error'

graphic list "Machine": 1 'Grafik_Verpackung_Step1_Blink-off'; 2 'Grafik_Verpackung_Step2'; 3 'Grafik_Verpackung_Blink-on'; 6..7 'Grafik_Verpackung_Step1_Blink-off'

screen "20_Messages" 800x480, template "01_One_Nav_Level"
   on GenerateScreen: SetTag("MainNavigationState", 2)
   AlarmView "Alarm view_1" at 0,104 size 800x375
   GraphicView "Graphic view_2" at 0,0 size 800x480; Picture "PopUpBackground"
      Visibility <- "PopUpBackground"

screen "30_Diagnostics" 800x480, template "01_One_Nav_Level"
   on GenerateScreen: SetTag("MainNavigationState", 3)
   SysDiagControl "System diagnostics view_1" at 0,104 size 800x375
   GraphicView "Graphic view_2" at 0,0 size 800x480; Picture "PopUpBackground"
      Visibility <- "PopUpBackground"

screen "40_Settings" 800x480, template "02_Settings"
   on GenerateScreen: SetTag("MainNavigationState", 4)
   Slider "Template_Slider_1" at 320,133 size 300x30; Caption 'SIMATIC'
      on Change: function_e4c2bb66("Brightness")
      ProcessValue <- "Brightness"
   TextField "Template_Text field_1" at 180,136 size 92x24; Text 'Brightness / Helligkeit'
   GraphicView "Graphic view_2" at 0,0 size 800x480; Picture "PopUpBackground"
      Visibility <- "PopUpBackground"

screen "10_Startscreen" 800x480, template "01_One_Nav_Level"
   on GenerateScreen: "GetStartScreenName"(); "CheckCurrentUserName"(); SetTag("MainNavigationState", 1)
   TextField "Text field_4" at 0,104 size 302x36; Text 'Short Conveyor'
   Group "Group" at 0,104 size 302x133
   Button "Button_3" at 58,150 size 96x32; TextOff 'Constant'
      on Click: InvertBit("Control_HMI_fromHMI_shortConveyor_constSpeedControl")
      Appearance <- "scConveyorShortConstSpeed_SetActive"
      ObjectEnable <- "scConveyorShortVarSpeed_SetActive"
   Button "Button_4" at 178,150 size 96x32; TextOff 'Variable'
      on Click: InvertBit("Control_HMI_fromHMI_shortConveyor_varSpeedControl")
      Appearance <- "scConveyorShortVarSpeed_SetActive"
      ObjectEnable <- "scConveyorShortConstSpeed_SetActive"
   IOField "I/O field_1" at 58,198 size 96x32; FormatPattern 999.99
      ObjectEnable <- "scConveyorShortConstSpeed_SetActive"
      ProcessValue <- "Control_HMI_fromHMI_shortConveyor_varSpeedPercentage"
   IOField "I/O field_2" at 178,198 size 96x32; FormatPattern 9.99999
      ProcessValue <- "scConveyorShortVarSpeed_SetSpeed"
   TextField "Text field_1" at 154,203 size 18x23; Text '%'
   TextField "Text field_2" at 274,203 size 28x23; Text 'm/s'
   TextField "Text field_3" at 2,203 size 53x23; Text 'Speed:'
   Group "Group_1" at 0,104 size 302x133
   Group "Group_6" at 0,234 size 302x133
   Group "Group_2" at 0,366 size 302x114
   Group "Group_3" at 302,104 size 255x175
   Group "Group_4" at 302,279 size 255x200
   Group "Group_7" at 557,324 size 243x156
   Group "Group_8" at 557,104 size 243x220
   TextField "Text field_12" at 0,234 size 302x36; Text 'Long Conveyor'
   Group "Group_5" at 0,234 size 302x133
   Button "Button_7" at 58,280 size 96x32; TextOff 'Constant'
      on Click: InvertBit("Control_HMI_fromHMI_longConveyor_constSpeedControl")
      Appearance <- "scConveyorLongConstSpeed_SetActive"
      ObjectEnable <- "scConveyorLongVarSpeed_SetActive"
   Button "Button_8" at 178,280 size 96x32; TextOff 'Variable'
      on Click: InvertBit("Control_HMI_fromHMI_longConveyor_varSpeedControl")
      Appearance <- "scConveyorLongVarSpeed_SetActive"
      ObjectEnable <- "scConveyorLongConstSpeed_SetActive"
   IOField "I/O field_6" at 58,328 size 96x32; FormatPattern 999.99
      ObjectEnable <- "scConveyorLongConstSpeed_SetActive"
      ProcessValue <- "Control_HMI_fromHMI_longConveyor_varSpeedPercentage"
   IOField "I/O field_7" at 178,328 size 96x32; FormatPattern 9.99999
      ProcessValue <- "scConveyorLongVarSpeed_SetSpeed"
   TextField "Text field_13" at 154,333 size 18x23; Text '%'
   TextField "Text field_14" at 274,333 size 28x23; Text 'm/s'
   TextField "Text field_15" at 2,333 size 53x23; Text 'Speed:'
   TextField "Text field_24" at 0,366 size 302x36; Text 'Workpiece Generation'
   Button "Button_6" at 58,436 size 96x32; TextOff 'Activate'
      on Click: InvertBit("Control_HMI_fromHMI_generateWorkpieces")
      Appearance <- "Control_HMI_fromHMI_generateWorkpieces"
   TextField "Text field_25" at 184,403 size 39x23; Text 'Cube'
   TextField "Text field_26" at 237,403 size 58x23; Text 'Cylinder'
   Circle "Circle_7" at 180,428 size 48x48
      Appearance <- "osWorkpieceCube_SetActive"
   Circle "Circle_8" at 242,428 size 48x48
      Appearance <- "osWorkpieceCylinder_SetActive"
   TextField "Text field_20" at 302,104 size 255x36; Text 'Piece Count'
   TextField "Text field_21" at 336,157 size 84x23; Text 'Workpieces'
   TextField "Text field_22" at 350,198 size 70x23; Text 'Cylindrical'
   TextField "Text field_23" at 381,240 size 39x23; Text 'Cube'
   IOField "I/O field_4" at 422,152 size 96x32; FormatPattern 99999
      ProcessValue <- "Control_HMI_toHMI_numWorkpieces"
   IOField "I/O field_5" at 422,193 size 96x32; FormatPattern 99999
      ProcessValue <- "Control_HMI_toHMI_numCylinders"
   IOField "I/O field_8" at 422,235 size 96x32; FormatPattern 99999
      ProcessValue <- "Control_HMI_toHMI_numCubes"
   Button "Button_1" at 331,345 size 96x32; TextOff 'Reset'
      on Press: function_b14e0dd5("Control_HMI_fromHMI_resetSimulation", 0); ResetBit("Control_HMI_fromHMI_shortConveyor_constSpeedControl"); ResetBit("Control_HMI_fromHMI_shortConveyor_varSpeedControl"); SetTag("Control_HMI_fromHMI_shortConveyor_varSpeedPercentage", 0); ResetBit("Control_HMI_fromHMI_longConveyor_constSpeedControl"); ResetBit("Control_HMI_fromHMI_longConveyor_varSpeedControl"); SetTag("Control_HMI_fromHMI_longConveyor_varSpeedPercentage", 0); ResetBit("Control_HMI_fromHMI_generateWorkpieces")
      Appearance <- "Control_HMI_fromHMI_resetSimulation"
   Circle "Circle_6" at 464,336 size 48x48
      Appearance <- "Control_HMI_toHMI_resetStatus"
   TextField "Text field_17" at 464,314 size 48x23; Text 'Status'
   Circle "Circle_5" at 464,388 size 48x48
      Appearance <- "Control_HMI_toHMI_Error"
   TextField "Text field_18" at 391,400 size 36x23; Text 'Error'
   TextField "Text field_16" at 374,445 size 53x23; Text 'Error ID'
   IOField "I/O field_3" at 440,441 size 96x32; FormatPattern FFFF
      ProcessValue <- "Control_HMI_toHMI_ErrorID"
   TextField "Text field_19" at 302,279 size 255x36; Text 'Simulation'
   TextField "Text field_7" at 587,383 size 128x23; Text 'Cylinder Extended'
   TextField "Text field_8" at 588,435 size 129x23; Text 'Cylinder Retracted'
   TextField "Text field_10" at 557,324 size 243x36; Text 'Limit Switches'
   Circle "Circle_3" at 723,370 size 48x48
      Appearance <- "csLimitSwitchCylinderNotExtended_Activated"
   Circle "Circle_4" at 723,422 size 48x48
      Appearance <- "csLimitSwitchCylinderRetracted_Activated"
   Circle "Circle_9" at 693,155 size 48x48
      Appearance <- "csLightSensorWorkpiece_Detected"
   TextField "Text field_5" at 609,167 size 77x23; Text 'Workpiece'
   TextField "Text field_6" at 625,220 size 58x23; Text 'Cylinder'
   TextField "Text field_9" at 647,273 size 39x23; Text 'Cube'
   TextField "Text field_11" at 557,104 size 243x36; Text 'Light Sensors'
   Circle "Circle_1" at 693,208 size 48x48
      Appearance <- "csLightSensorCylinder_Detected"
   Circle "Circle_2" at 693,261 size 48x48
      Appearance <- "csLightSensorCube_Detected"

Template "02_Two_Nav_Levels" 800x480
   GraphicView "gfxPrevScreenIcon" at 760,444 size 24x24; Picture "PrevScreen_Icon"
   Button "btnSubNav1" at 0,432 size 120x48; TextOff 'Overview / Übersicht'
      on Click: SetTag("SubNavigationState", 1)
   Button "btnSubNav2" at 120,432 size 120x48; TextOff 'Module 1 / Modul 1'
      on Click: SetTag("SubNavigationState", 2)
   Button "btnSubNav3" at 240,432 size 120x48; TextOff 'Module 2 / Modul 2'
      on Click: SetTag("SubNavigationState", 3)
   Button "btnSubNav4" at 360,432 size 120x48; TextOff 'Module 3 / Modul 3'
      on Click: SetTag("SubNavigationState", 4)
   Button "btnSubNav5" at 480,432 size 120x48; TextOff 'Module 4 / Modul 4'
      on Click: SetTag("SubNavigationState", 5)
   Button "btnSubNav6" at 600,432 size 120x48; TextOff 'Module 5 / Modul 5'
      on Click: SetTag("SubNavigationState", 6)
   Button "btnPreviousScreen" at 744,432 size 56x48; TextOff 'Text'
      on Click: function_efd93a16()
   Gauge "gaugeDiagStateUpdate" at 566,2 size 50x50; CaptionText 'SIMATIC'
      on Change: "CheckDiagState"()
      ProcessValue <- "@DiagnosticsIndicatorTag"
   TextField "txtTitleBar" at 16,8 size 495x32; Text 'Sorting Plant / Applikation'
   GraphicView "gfxNavigationIcon" at 761,15 size 23x19; Picture "Hamburger_Icon"
   Button "btnNavigation" at 744,0 size 56x48; TextOff 'Text'
      on Click: function_cf6f4242("GraphX_Slidein_Right", 1)
   TextField "txtStateHeadline" at 75,55 size 123x23; Text 'State / Status'
   TextField "txtRecipeHeadline" at 281,55 size 154x23; Text 'Current Recipe / Rezeptur'
   TextField "txtOperatorHeadline" at 527,55 size 129x23; Text 'Operator / Bediener'
   SymbolicIOField "ioState" at 75,72 size 119x30; TextOn '1'; TextOff '0'; TextList "Machine State"
      ProcessValue <- "CurrentMachineState"
   IOField "ioRecipe" at 281,72 size 158x30; FormatPattern ??????????????????????????????
      ProcessValue <- "CurrentRecipeName"
   IOField "ioOperator" at 527,72 size 126x30; FormatPattern ??????????????????
      ProcessValue <- "CurrentUserName"
   Button "btnState" at 202,56 size 40x40; TextOff '...'; PictureOff "More_Icon"
      on Click: "ShowOperatingModePopUp"()
   Button "btnRecipe" at 449,56 size 40x40; TextOff '...'; PictureOff "More_Icon"
      on Click: "ShowRecipePopUp"()
   Rectangle "rectState" at 0,48 size 56x56
      Appearance <- "CurrentMachineState"
   Rectangle "rectSystemDiagnosticsIndicator" at 744,48 size 56x56
      Appearance <- "DiagState"
   GraphicIOField "gioDiagState" at 756,60 size 32x32; PictureList "DiagState_3"
      ProcessValue <- "DiagState"
   Button "btnDiagState" at 744,48 size 56x56; TextOff 'Text'
      on Click: ActivateScreen("30_Diagnostics", 0)
   Button "btnOperator" at 669,56 size 40x40; TextOff '...'; PictureOff "More_Icon"
      on Click: "ShowLoginPopUp"()
   Button "btnStartscreen" at 0,0 size 250x45; TextOff 'Text'
      on Click: "ActivateStartScreen"()
   Button "btnSubNavActive1" at 0,432 size 120x48; TextOff 'Overview / Übersicht'
      Visibility <- "SubNavigationState"
   Button "btnSubNavActive2" at 120,432 size 120x48; TextOff 'Module 1 / Modul 1'
      Visibility <- "SubNavigationState"
   Button "btnSubNavActive3" at 240,432 size 120x48; TextOff 'Module 2 / Modul 2'
      Visibility <- "SubNavigationState"
   Button "btnSubNavActive4" at 360,432 size 120x48; TextOff 'Module 3 / Modul 3'
      Visibility <- "SubNavigationState"
   Button "btnSubNavActive5" at 480,432 size 120x48; TextOff 'Module 4 / Modul 4'
      Visibility <- "SubNavigationState"
   Button "btnSubNavActive6" at 600,432 size 120x48; TextOff 'Module 5 / Modul 5'
      Visibility <- "SubNavigationState"
   Rectangle "rectIndicatorActive1" at 0,475 size 120x5
      Visibility <- "SubNavigationState"
   Rectangle "rectIndicatorActive2" at 120,475 size 120x5
      Visibility <- "SubNavigationState"
   Rectangle "rectIndicatorActive3" at 240,475 size 120x5
      Visibility <- "SubNavigationState"
   Rectangle "rectIndicatorActive4" at 360,475 size 120x5
      Visibility <- "SubNavigationState"
   Rectangle "rectIndicatorActive5" at 480,475 size 120x5
      Visibility <- "SubNavigationState"
   Rectangle "rectIndicatorActive6" at 600,475 size 120x5
      Visibility <- "SubNavigationState"

Template "03_Three_Nav_Levels" 800x480
   Button "btnStartscreen" at 0,0 size 326x45; TextOff 'Text'
      on Click: "ActivateStartScreen"()
   Gauge "gaugeDiagStateUpdate" at 566,2 size 50x50; CaptionText 'SIMATIC'
      on Change: "CheckDiagState"()
      ProcessValue <- "@DiagnosticsIndicatorTag"
   TextField "txtTitleBar" at 16,8 size 495x32; Text 'Sorting Plant / Applikation'
   GraphicView "gfxNavigationIcon" at 761,15 size 23x19; Picture "Hamburger_Icon"
   Button "btnNavigation" at 744,0 size 56x48; TextOff 'Text'
      on Click: function_cf6f4242("GraphX_Slidein_Right", 1)
   Rectangle "rectSystemDiagnosticsIndicator" at 744,48 size 56x56
      Appearance <- "DiagState"
   GraphicIOField "gioDiagState" at 756,60 size 32x32; PictureList "DiagState_3"
      ProcessValue <- "DiagState"
   Button "btnDiagState" at 744,48 size 56x56; TextOff 'Text'
      on Click: ActivateScreen("30_Diagnostics", 0)
   TextField "txtStateHeadline" at 75,55 size 123x23; Text 'State / Status'
   TextField "txtOperatorHeadline" at 527,55 size 129x23; Text 'Operator / Bediener'
   SymbolicIOField "ioState" at 75,72 size 119x30; TextOn '1'; TextOff '0'; TextList "Machine State"
      ProcessValue <- "CurrentMachineState"
   IOField "ioOperator" at 527,72 size 126x30; FormatPattern ??????????????????
      ProcessValue <- "CurrentUserName"
   Button "btnState" at 202,56 size 40x40; TextOff '...'; PictureOff "More_Icon"
      on Click: "ShowOperatingModePopUp"()
   Button "btnOperator" at 669,56 size 40x40; TextOff '...'; PictureOff "More_Icon"
      on Click: "ShowLoginPopUp"()
   Rectangle "rectState" at 0,48 size 56x56
      Appearance <- "CurrentMachineState"
   TextField "txtRecipeHeadline" at 281,55 size 154x23; Text 'Current Recipe / Rezeptur'
   IOField "ioRecipe" at 281,72 size 158x30; FormatPattern ??????????????????????????????
      ProcessValue <- "CurrentRecipeName"
   Button "btnRecipe" at 449,56 size 40x40; TextOff '...'; PictureOff "More_Icon"
      on Click: "ShowRecipePopUp"()
   Button "btnThirdLevel4btnOff1" at 0,104 size 56x83; TextOff 'Text'
   Button "btnThirdLevel4btnOff2" at 0,186 size 56x83; TextOff 'Text'
   Button "btnThirdLevel4btnOff3" at 0,268 size 56x83; TextOff 'Text'
   Button "btnThirdLevel4btnOff4" at 0,350 size 56x82; TextOff 'Text'
   Button "btnThirdLevel4btnOn1" at 0,187 size 56x81; TextOff 'Text'
      Visibility <- "ThirdLevelNavigationState"
   Button "btnThirdLevel4btnOn2" at 0,104 size 56x82; TextOff 'Text'
      Visibility <- "ThirdLevelNavigationState"
   Button "btnThirdLevel4btnOn3" at 0,269 size 56x81; TextOff 'Text'
      Visibility <- "ThirdLevelNavigationState"
   Button "btnThirdLevel4btnOn4" at 0,351 size 56x81; TextOff 'Text'
      Visibility <- "ThirdLevelNavigationState"
   Rectangle "rectIndicator4btnActive1" at 0,104 size 5x82
      Visibility <- "ThirdLevelNavigationState"
   Rectangle "rectIndicator4btnActive2" at 0,187 size 5x81
      Visibility <- "ThirdLevelNavigationState"
   Rectangle "rectIndicator4btnActive3" at 0,269 size 5x81
      Visibility <- "ThirdLevelNavigationState"
   Rectangle "rectIndicator4btnActive4" at 0,351 size 5x81
      Visibility <- "ThirdLevelNavigationState"
   Button "btnSubNav1" at 0,432 size 120x48; TextOff 'Overview / Übersicht'
      on Click: SetTag("SubNavigationState", 1)
   Button "btnSubNav2" at 120,432 size 120x48; TextOff 'Module 1 / Modul 1'
      on Click: SetTag("SubNavigationState", 2)
   Button "btnSubNav3" at 240,432 size 120x48; TextOff 'Module 2 / Modul 2'
      on Click: SetTag("SubNavigationState", 3)
   Button "btnSubNav4" at 360,432 size 120x48; TextOff 'Module 3 / Modul 3'
      on Click: SetTag("SubNavigationState", 4)
   Button "btnSubNav5" at 480,432 size 120x48; TextOff 'Module 4 / Modul 4'
      on Click: SetTag("SubNavigationState", 5)
   Button "btnSubNav6" at 600,432 size 120x48; TextOff 'Module 5 / Modul 5'
      on Click: SetTag("SubNavigationState", 6)
   GraphicView "gfxPrevScreenIcon" at 760,444 size 24x24; Picture "PrevScreen_Icon"
   Button "btnPreviousScreen" at 744,432 size 56x48; TextOff 'Text'
      on Click: function_efd93a16()
   Button "btnSubNavActive1" at 0,432 size 120x48; TextOff 'Overview / Übersicht'
      Visibility <- "SubNavigationState"
   Button "btnSubNavActive2" at 120,432 size 120x48; TextOff 'Module 1 / Modul 1'
      Visibility <- "SubNavigationState"
   Button "btnSubNavActive3" at 240,432 size 120x48; TextOff 'Module 2 / Modul 2'
      Visibility <- "SubNavigationState"
   Button "btnSubNavActive4" at 360,432 size 120x48; TextOff 'Module 3 / Modul 3'
      Visibility <- "SubNavigationState"
   Button "btnSubNavActive5" at 480,432 size 120x48; TextOff 'Module 4 / Modul 4'
      Visibility <- "SubNavigationState"
   Button "btnSubNavActive6" at 600,432 size 120x48; TextOff 'Module 5 / Modul 5'
      Visibility <- "SubNavigationState"
   Rectangle "rectIndicatorActive1" at 0,475 size 120x5
      Visibility <- "SubNavigationState"
   Rectangle "rectIndicatorActive2" at 120,475 size 120x5
      Visibility <- "SubNavigationState"
   Rectangle "rectIndicatorActive3" at 240,475 size 120x5
      Visibility <- "SubNavigationState"
   Rectangle "rectIndicatorActive4" at 360,475 size 120x5
      Visibility <- "SubNavigationState"
   Rectangle "rectIndicatorActive5" at 480,475 size 120x5
      Visibility <- "SubNavigationState"
   Rectangle "rectIndicatorActive6" at 600,475 size 120x5
      Visibility <- "SubNavigationState"

Template "03_Three_Nav_Levels_w_OptionPanel" 800x480
   Button "btnStartscreen" at 0,0 size 326x45; TextOff 'Text'
      on Click: "ActivateStartScreen"()
   Gauge "gaugeDiagStateUpdate" at 566,2 size 50x50; CaptionText 'SIMATIC'
      on Change: "CheckDiagState"()
      ProcessValue <- "@DiagnosticsIndicatorTag"
   TextField "txtTitleBar" at 16,8 size 495x32; Text 'Sorting Plant / Applikation'
   GraphicView "gfxNavigationIcon" at 761,15 size 23x19; Picture "Hamburger_Icon"
   Button "btnNavigation" at 744,0 size 56x48; TextOff 'Text'
      on Click: function_cf6f4242("GraphX_Slidein_Right", 1)
   Rectangle "rectSystemDiagnosticsIndicator" at 744,48 size 56x56
      Appearance <- "DiagState"
   GraphicIOField "gioDiagState" at 756,60 size 32x32; PictureList "DiagState_3"
      ProcessValue <- "DiagState"
   Button "btnDiagState" at 744,48 size 56x56; TextOff 'Text'
      on Click: ActivateScreen("30_Diagnostics", 0)
   TextField "txtStateHeadline" at 75,55 size 123x23; Text 'State / Status'
   TextField "txtOperatorHeadline" at 527,55 size 129x23; Text 'Operator / Bediener'
   SymbolicIOField "ioState" at 75,72 size 119x30; TextOn '1'; TextOff '0'; TextList "Machine State"
      ProcessValue <- "CurrentMachineState"
   IOField "ioOperator" at 527,72 size 126x30; FormatPattern ??????????????????
      ProcessValue <- "CurrentUserName"
   Button "btnState" at 202,56 size 40x40; TextOff '...'; PictureOff "More_Icon"
      on Click: "ShowOperatingModePopUp"()
   Button "btnOperator" at 669,56 size 40x40; TextOff '...'; PictureOff "More_Icon"
      on Click: "ShowLoginPopUp"()
   Rectangle "rectState" at 0,48 size 56x56
      Appearance <- "CurrentMachineState"
   TextField "txtRecipeHeadline" at 281,55 size 154x23; Text 'Current Recipe / Rezeptur'
   IOField "ioRecipe" at 281,72 size 158x30; FormatPattern ??????????????????????????????
      ProcessValue <- "CurrentRecipeName"
   Button "btnRecipe" at 449,56 size 40x40; TextOff '...'; PictureOff "More_Icon"
      on Click: "ShowRecipePopUp"()
   Button "btnThirdLevelOff1" at 0,104 size 56x83; TextOff 'Text'
   Button "btnThirdLevelOff2" at 0,186 size 56x83; TextOff 'Text'
   Button "btnThirdLevelOff3" at 0,268 size 56x83; TextOff 'Text'
   Button "btnThirdLevelOff4" at 0,350 size 56x82; TextOff 'Text'
   Button "btnThirdLevelOn1" at 0,187 size 56x81; TextOff 'Text'
      Visibility <- "ThirdLevelNavigationState"
   Button "btnThirdLevelOn2" at 0,104 size 56x82; TextOff 'Text'
      Visibility <- "ThirdLevelNavigationState"
   Button "btnThirdLevelOn3" at 0,269 size 56x81; TextOff 'Text'
      Visibility <- "ThirdLevelNavigationState"
   Button "btnThirdLevelOn4" at 0,351 size 56x81; TextOff 'Text'
      Visibility <- "ThirdLevelNavigationState"
   Rectangle "rectIndicatorActive1_1" at 0,104 size 5x82
      Visibility <- "ThirdLevelNavigationState"
   Rectangle "rectIndicatorActive1_2" at 0,187 size 5x81
      Visibility <- "ThirdLevelNavigationState"
   Rectangle "rectIndicatorActive1_3" at 0,269 size 5x81
      Visibility <- "ThirdLevelNavigationState"
   Rectangle "rectIndicatorActive1_4" at 0,351 size 5x81
      Visibility <- "ThirdLevelNavigationState"
   Button "btnOption1btn1" at 744,104 size 56x328; TextOff 'Text'; PictureOff "ManFunctions_Off"; PictureOn "ManFunctions_Off"
      on Click: "ShowOptionPanelPopUp"()
   Button "btnSubNav1" at 0,432 size 120x48; TextOff 'Overview / Übersicht'
      on Click: SetTag("SubNavigationState", 1)
   Button "btnSubNav2" at 120,432 size 120x48; TextOff 'Module 1 / Modul 1'
      on Click: SetTag("SubNavigationState", 2)
   Button "btnSubNav3" at 240,432 size 120x48; TextOff 'Module 2 / Modul 2'
      on Click: SetTag("SubNavigationState", 3)
   Button "btnSubNav4" at 360,432 size 120x48; TextOff 'Module 3 / Modul 3'
      on Click: SetTag("SubNavigationState", 4)
   Button "btnSubNav5" at 480,432 size 120x48; TextOff 'Module 4 / Modul 4'
      on Click: SetTag("SubNavigationState", 5)
   Button "btnSubNav6" at 600,432 size 120x48; TextOff 'Module 5 / Modul 5'
      on Click: SetTag("SubNavigationState", 6)
   GraphicView "gfxPrevScreenIcon" at 760,444 size 24x24; Picture "PrevScreen_Icon"
   Button "btnPreviousScreen" at 744,432 size 56x48; TextOff 'Text'
      on Click: function_efd93a16()
   Button "btnSubNavActive1" at 0,432 size 120x48; TextOff 'Overview / Übersicht'
      Visibility <- "SubNavigationState"
   Button "btnSubNavActive2" at 120,432 size 120x48; TextOff 'Module 1 / Modul 1'
      Visibility <- "SubNavigationState"
   Button "btnSubNavActive3" at 240,432 size 120x48; TextOff 'Module 2 / Modul 2'
      Visibility <- "SubNavigationState"
   Button "btnSubNavActive4" at 360,432 size 120x48; TextOff 'Module 3 / Modul 3'
      Visibility <- "SubNavigationState"
   Button "btnSubNavActive5" at 480,432 size 120x48; TextOff 'Module 4 / Modul 4'
      Visibility <- "SubNavigationState"
   Button "btnSubNavActive6" at 600,432 size 120x48; TextOff 'Module 5 / Modul 5'
      Visibility <- "SubNavigationState"
   Rectangle "rectIndicatorActive1" at 0,475 size 120x5
      Visibility <- "SubNavigationState"
   Rectangle "rectIndicatorActive2" at 120,475 size 120x5
      Visibility <- "SubNavigationState"
   Rectangle "rectIndicatorActive3" at 240,475 size 120x5
      Visibility <- "SubNavigationState"
   Rectangle "rectIndicatorActive4" at 360,475 size 120x5
      Visibility <- "SubNavigationState"
   Rectangle "rectIndicatorActive5" at 480,475 size 120x5
      Visibility <- "SubNavigationState"
   Rectangle "rectIndicatorActive6" at 600,475 size 120x5
      Visibility <- "SubNavigationState"

Template "01_One_Nav_Level" 800x480
   Rectangle "rectSystemDiagnosticsIndicator" at 744,48 size 56x56
      Appearance <- "DiagState"
   GraphicIOField "gioDiagState" at 756,60 size 32x32; PictureList "DiagState_3"
      ProcessValue <- "DiagState"
   Button "btnDiagState" at 744,48 size 56x56; TextOff 'Text'
      on Click: ActivateScreen("30_Diagnostics", 0)
   TextField "txtStateHeadline" at 75,55 size 123x23; Text 'State / Status'
   TextField "txtOperatorHeadline" at 527,55 size 129x23; Text 'Operator / Bediener'
   SymbolicIOField "ioState" at 75,72 size 119x30; TextOn '1'; TextOff '0'; TextList "Machine State"
      ProcessValue <- "CurrentMachineState"
   IOField "ioOperator" at 527,72 size 126x30; FormatPattern ??????????????????
      ProcessValue <- "CurrentUserName"
   Button "btnState" at 202,56 size 40x40; TextOff '...'; PictureOff "More_Icon"
      on Click: "ShowOperatingModePopUp"()
   Button "btnOperator" at 669,56 size 40x40; TextOff '...'; PictureOff "More_Icon"
      on Click: "ShowLoginPopUp"()
   Rectangle "rectState" at 0,48 size 56x56
      Appearance <- "CurrentMachineState"
   TextField "txtRecipeHeadline" at 281,55 size 154x23; Text 'Current Recipe / Rezeptur'
   IOField "ioRecipe" at 281,72 size 158x30; FormatPattern ??????????????????????????????
      ProcessValue <- "CurrentRecipeName"
   Button "btnRecipe" at 449,56 size 40x40; TextOff '...'; PictureOff "More_Icon"
      on Click: "ShowRecipePopUp"()
   Gauge "gaugeDiagStateUpdate" at 566,2 size 50x50; CaptionText 'SIMATIC'
      on Change: "CheckDiagState"()
      ProcessValue <- "@DiagnosticsIndicatorTag"
   GraphicView "gfxNavigationIcon" at 761,15 size 23x19; Picture "Hamburger_Icon"
   Button "btnNavigation" at 744,0 size 56x48; TextOff 'Text'
      on Click: function_cf6f4242("GraphX_Slidein_Right", 1)
   TextField "txtTitleBar" at 16,8 size 495x32; Text 'Sorting Plant / Applikation'
   Button "btnStartscreen" at 0,0 size 250x45; TextOff 'Text'
      on Click: "ActivateStartScreen"()

Template "02_Two_Nav_Levels_Large_Text" 800x480
   Gauge "gaugeDiagStateUpdate" at 566,2 size 50x50; CaptionText 'SIMATIC'
      on Change: "CheckDiagState"()
      ProcessValue <- "@DiagnosticsIndicatorTag"
   TextField "txtTitleBar" at 16,8 size 495x32; Text 'Sorting Plant / Applikation'
   GraphicView "gfxNavigationIcon" at 761,15 size 23x19; Picture "Hamburger_Icon"
   Button "btnNavigation" at 744,0 size 56x48; TextOff 'Text'
      on Click: function_cf6f4242("GraphX_Slidein_Right", 1)
   TextField "txtStateHeadline" at 75,55 size 123x23; Text 'State / Status'
   TextField "txtRecipeHeadline" at 281,55 size 154x23; Text 'Current Recipe / Rezeptur'
   TextField "txtOperatorHeadline" at 527,55 size 129x23; Text 'Operator / Bediener'
   SymbolicIOField "ioState" at 75,72 size 119x30; TextOn '1'; TextOff '0'; TextList "Machine State"
      ProcessValue <- "CurrentMachineState"
   IOField "ioRecipe" at 281,72 size 158x30; FormatPattern ??????????????????????????????
      ProcessValue <- "CurrentRecipeName"
   IOField "ioOperator" at 527,72 size 126x30; FormatPattern ??????????????????
      ProcessValue <- "CurrentUserName"
   Button "btnState" at 202,56 size 40x40; TextOff '...'; PictureOff "More_Icon"
      on Click: "ShowOperatingModePopUp"()
   Button "btnRecipe" at 449,56 size 40x40; TextOff '...'; PictureOff "More_Icon"
      on Click: "ShowRecipePopUp"()
   Rectangle "rectState" at 0,48 size 56x56
      Appearance <- "CurrentMachineState"
   GraphicView "gfxPrevScreenIcon" at 760,444 size 24x24; Picture "PrevScreen_Icon"
   Button "btnPreviousScreen" at 744,432 size 56x48; TextOff 'Text'
      on Click: function_efd93a16()
   TextField "txtCurrentStateInfo" at 16,444 size 505x24; Text 'Optional Text about current state / Optional. Text aktueller Status'
   Rectangle "rectSystemDiagnosticsIndicator" at 744,48 size 56x56
      Appearance <- "DiagState"
   GraphicIOField "gioDiagState" at 756,60 size 32x32; PictureList "DiagState_3"
      ProcessValue <- "DiagState"
   Button "btnDiagState" at 744,48 size 56x56; TextOff 'Text'
      on Click: ActivateScreen("30_Diagnostics", 0)
   Button "btnOperator" at 669,56 size 40x40; TextOff '...'; PictureOff "More_Icon"
      on Click: "ShowLoginPopUp"()
   Button "btnStartscreen" at 0,0 size 250x45; TextOff 'Text'
      on Click: "ActivateStartScreen"()
   Rectangle "rectSubNavigation1" at 0,104 size 264x83
      Appearance <- "ThirdLevelNavigationState"
   Rectangle "rectSubNavigation2" at 0,186 size 264x83
      Appearance <- "ThirdLevelNavigationState"
   Rectangle "rectSubNavigation3" at 0,268 size 264x83
      Appearance <- "ThirdLevelNavigationState"
   Rectangle "rectSubNavigation4" at 0,350 size 264x82
      Appearance <- "ThirdLevelNavigationState"
   TextField "txtOption1" at 16,120 size 232x24; Text 'Option 1'
   IOField "ioValueOption1" at 16,152 size 236x24; FormatPattern ??????????????????????????????????????????????????
   TextField "txtOption2" at 16,202 size 232x24; Text 'Option 2'
   IOField "ioValueOption2" at 16,234 size 236x24; FormatPattern ??????????????????????????????????????????????????
   TextField "txtOption3" at 16,284 size 232x24; Text 'Option 3'
   IOField "ioValueOption3" at 16,316 size 236x24; FormatPattern ??????????????????????????????????????????????????
   TextField "txtOption4" at 16,366 size 232x24; Text 'Option 4'
   IOField "ioValueOption4" at 16,398 size 236x24; FormatPattern ??????????????????????????????????????????????????
   Button "btnSubNavigation1" at 0,104 size 264x83; TextOff 'Text'
      on Click: SetTag("ThirdLevelNavigationState", 1)
   Button "btnSubNavigation2" at 0,186 size 264x83; TextOff 'Text'
      on Click: SetTag("ThirdLevelNavigationState", 2)
   Button "btnSubNavigation3" at 0,268 size 264x83; TextOff 'Text'
      on Click: SetTag("ThirdLevelNavigationState", 3)
   Button "btnSubNavigation4" at 0,350 size 264x83; TextOff 'Text'
      on Click: SetTag("ThirdLevelNavigationState", 4)

Template "02_Two_Nav_Levels_Text" 800x480
   Button "btnSubNav1" at 0,120 size 136x56; TextOn 'Item 1'; TextOff 'Item 1'
      on Click: SetTag("SubNavigationState", 1)
   Button "btnSubNav2" at 0,175 size 136x56; TextOn 'Item 2'; TextOff 'Item 2'
      on Click: SetTag("SubNavigationState", 2)
   Button "btnSubNav3" at 0,230 size 136x60; TextOn 'Item 3'; TextOff 'Item 3'
      on Click: SetTag("SubNavigationState", 3)
   GraphicView "gfxRuntimeStop" at 57,443 size 23x28; Picture "Power_dark"
   Button "btnRuntimeStop" at 0,432 size 136x48; TextOff 'Text'
      on Click: StopRuntime(0)
   Button "btnSubNav3_1" at 0,289 size 136x60; TextOn 'Item 4'; TextOff 'Item 4'
      on Click: SetTag("SubNavigationState", 4)
   Button "btnSubNav3_2" at 0,348 size 136x60; TextOn 'Item 5'; TextOff 'Item 5'
      on Click: SetTag("SubNavigationState", 5)
   Button "btnSubNavActive3" at 0,230 size 136x60; TextOff 'Item 3'
      Visibility <- "SubNavigationState"
   Button "btnSubNavActive1" at 0,120 size 136x56; TextOff 'Item 1'
      Visibility <- "SubNavigationState"
   Button "btnSubNavActive2" at 0,175 size 136x56; TextOff 'Item 2'
      Visibility <- "SubNavigationState"
   Rectangle "rectIndicatorActive3" at 0,230 size 5x60
      Visibility <- "SubNavigationState"
   Rectangle "rectIndicatorActive1" at 0,120 size 5x56
      Visibility <- "SubNavigationState"
   Rectangle "rectIndicatorActive2" at 0,175 size 5x56
      Visibility <- "SubNavigationState"
   Button "btnSubNavActive3_1" at 0,290 size 136x60; TextOff 'Item 4'
      Visibility <- "SubNavigationState"
   Rectangle "rectIndicatorActive3_1" at 0,290 size 5x60
      Visibility <- "SubNavigationState"
   Button "btnSubNavActive3_2" at 0,350 size 136x60; TextOff 'Item 5'
      Visibility <- "SubNavigationState"
   Rectangle "rectIndicatorActive3_2" at 0,350 size 5x60
      Visibility <- "SubNavigationState"
   Gauge "gaugeDiagStateUpdate" at 566,2 size 50x50; CaptionText 'SIMATIC'
      on Change: "CheckDiagState"()
      ProcessValue <- "@DiagnosticsIndicatorTag"
   GraphicView "gfxNavigationIcon" at 761,15 size 23x19; Picture "Hamburger_Icon"
   Button "btnNavigation" at 744,0 size 56x48; TextOff 'Text'
      on Click: function_cf6f4242("GraphX_Slidein_Right", 1)
   TextField "txtTitleBar" at 16,8 size 495x32; Text 'Sorting Plant / Applikation'
   Button "btnStartscreen" at 0,0 size 250x45; TextOff 'Text'
      on Click: "ActivateStartScreen"()
   TextField "txtStateHeadline" at 75,55 size 123x23; Text 'State / Status'
   TextField "txtOperatorHeadline" at 527,55 size 129x23; Text 'Operator / Bediener'
   SymbolicIOField "ioState" at 75,72 size 119x30; TextOn '1'; TextOff '0'; TextList "Machine State"
      ProcessValue <- "CurrentMachineState"
   IOField "ioOperator" at 527,72 size 126x30; FormatPattern ??????????????????
      ProcessValue <- "CurrentUserName"
   Button "btnState" at 202,56 size 40x40; TextOff '...'; PictureOff "More_Icon"
      on Click: "ShowOperatingModePopUp"()
   Button "btnOperator" at 669,56 size 40x40; TextOff '...'; PictureOff "More_Icon"
      on Click: "ShowLoginPopUp"()
   Rectangle "rectState" at 0,48 size 56x56
      Appearance <- "CurrentMachineState"
   TextField "txtRecipeHeadline" at 281,55 size 154x23; Text 'Current Recipe / Rezeptur'
   IOField "ioRecipe" at 281,72 size 158x30; FormatPattern ??????????????????????????????
      ProcessValue <- "CurrentRecipeName"
   Button "btnRecipe" at 449,56 size 40x40; TextOff '...'; PictureOff "More_Icon"
      on Click: "ShowRecipePopUp"()
   Rectangle "rectSystemDiagnosticsIndicator" at 744,48 size 56x56
      Appearance <- "DiagState"
   GraphicIOField "gioDiagState" at 756,60 size 32x32; PictureList "DiagState_3"
      ProcessValue <- "DiagState"
   Button "btnDiagState" at 744,48 size 56x56; TextOff 'Text'
      on Click: ActivateScreen("30_Diagnostics", 0)

Template "02_Settings" 800x480
   Button "btnSubNav1" at 0,120 size 136x56; TextOn 'Display'; TextOff 'Display'
      on Click: SetTag("SubNavigationState", 1)
   GraphicView "gfxRuntimeStop" at 57,443 size 23x28; Picture "Power_dark"
   Button "btnRuntimeStop" at 0,432 size 136x48; TextOff 'Text'
      on Click: StopRuntime(0)
   Button "btnSubNavActive1" at 0,120 size 136x56; TextOn 'Display'; TextOff 'Display'
      Visibility <- "SubNavigationState"
   Rectangle "rectIndicatorActive1" at 0,120 size 5x56
      Visibility <- "SubNavigationState"
   Gauge "gaugeDiagStateUpdate" at 566,2 size 50x50; CaptionText 'SIMATIC'
      on Change: "CheckDiagState"()
      ProcessValue <- "@DiagnosticsIndicatorTag"
   GraphicView "gfxNavigationIcon" at 761,15 size 23x19; Picture "Hamburger_Icon"
   Button "btnNavigation" at 744,0 size 56x48; TextOff 'Text'
      on Click: function_cf6f4242("GraphX_Slidein_Right", 1)
   TextField "txtTitleBar" at 16,8 size 495x32; Text 'Sorting Plant / Applikation'
   Button "btnStartscreen" at 0,0 size 250x45; TextOff 'Text'
      on Click: "ActivateStartScreen"()
   TextField "txtStateHeadline" at 75,55 size 123x23; Text 'State / Status'
   TextField "txtOperatorHeadline" at 527,55 size 129x23; Text 'Operator / Bediener'
   SymbolicIOField "ioState" at 75,72 size 119x30; TextOn '1'; TextOff '0'; TextList "Machine State"
      ProcessValue <- "CurrentMachineState"
   IOField "ioOperator" at 527,72 size 126x30; FormatPattern ??????????????????
      ProcessValue <- "CurrentUserName"
   Button "btnState" at 202,56 size 40x40; TextOff '...'; PictureOff "More_Icon"
      on Click: "ShowOperatingModePopUp"()
   Button "btnOperator" at 669,56 size 40x40; TextOff '...'; PictureOff "More_Icon"
      on Click: "ShowLoginPopUp"()
   Rectangle "rectState" at 0,48 size 56x56
      Appearance <- "CurrentMachineState"
   TextField "txtRecipeHeadline" at 281,55 size 154x23; Text 'Current Recipe / Rezeptur'
   IOField "ioRecipe" at 281,72 size 158x30; FormatPattern ??????????????????????????????
      ProcessValue <- "CurrentRecipeName"
   Button "btnRecipe" at 449,56 size 40x40; TextOff '...'; PictureOff "More_Icon"
      on Click: "ShowRecipePopUp"()
   Rectangle "rectSystemDiagnosticsIndicator" at 744,48 size 56x56
      Appearance <- "DiagState"
   GraphicIOField "gioDiagState" at 756,60 size 32x32; PictureList "DiagState_3"
      ProcessValue <- "DiagState"
   Button "btnDiagState" at 744,48 size 56x56; TextOff 'Text'
      on Click: ActivateScreen("30_Diagnostics", 0)

PopupScreen "Template_Logon" 320x352
   on ClearScreen: ResetBit("PopUpBackground")
   on GenerateScreen: SetBit("PopUpBackground")
   TextField "Template_Text field_1" at 16,0 size 215x40; Text 'Login'
   Button "Button_2" at 16,240 size 288x40; TextOn 'LOGIN / ANMELDEN'; TextOff 'LOGIN / ANMELDEN'
      on Click: function_a9b89908("Password", "UserName"); function_efd93a16("Template_Logon", 0, 0, 0, -1, 1)
   IOField "I/O field_1" at 16,84 size 288x40; FormatPattern ??????????????????????????????
      ProcessValue <- "UserName"
   TextField "Text field_1" at 16,56 size 288x24; Text 'User Name / Name'
   IOField "I/O field_2" at 16,168 size 288x40; FormatPattern ??????????????????????????????
      ProcessValue <- "Password"
   TextField "Text field_2" at 16,140 size 288x24; Text 'Password / Passwort'
   Button "Button_1" at 16,296 size 288x40; TextOn 'CLOSE / SCHLIESSEN'; TextOff 'CLOSE / SCHLIESSEN'
      on Click: function_efd93a16("Template_Logon", 0, 0, 0, -1, 1)
      on Press: function_b14e0dd5("ButtonDown", 0)
      Appearance <- "ButtonDown"

PopupScreen "Template_Logon_Logoff" 320x352
   on ClearScreen: ResetBit("PopUpBackground")
   on GenerateScreen: SetBit("PopUpBackground")
   TextField "Template_Text field_1" at 16,0 size 215x40; Text 'Login'
   Button "Button_2" at 16,240 size 136x40; TextOn 'LOG OFF / ABMELDEN'; TextOff 'LOG OFF / ABMELDEN'
      on Click: function_f23ef4c9()
   IOField "I/O field_1" at 16,84 size 288x40; FormatPattern ??????????????????????????????
      ProcessValue <- "UserName"
   TextField "Text field_1" at 16,56 size 288x24; Text 'User Name / Name'
   IOField "I/O field_2" at 16,168 size 288x40; FormatPattern ??????????????????????????????
      ProcessValue <- "Password"
   TextField "Text field_2" at 16,140 size 288x24; Text 'Password / Passwort'
   Button "Button_1" at 16,296 size 288x40; TextOn 'CLOSE / SCHLIESSEN'; TextOff 'CLOSE / SCHLIESSEN'
      on Click: function_efd93a16("Template_Logon_Logoff", 0, 0, 0, -1, 1)
      on Press: function_b14e0dd5("ButtonDown", 0)
      Appearance <- "ButtonDown"
   Button "Button_3" at 168,240 size 136x40; TextOn 'LOGIN / ANMELDEN'; TextOff 'LOGIN / ANMELDEN'
      on Click: function_a9b89908("Password", "UserName"); function_efd93a16("Template_Logon_Logoff", 0, 0, 0, -1, 1)

PopupScreen "Template_Operating_Mode" 424x360
   on ClearScreen: ResetBit("PopUpBackground")
   on GenerateScreen: SetBit("PopUpBackground")
   TextField "Template_Text field_1" at 14,0 size 336x40; Text 'Operating Mode / Betriebsmodus'
   Button "Button_1" at 80,304 size 260x40; TextOn 'CLOSE / SCHLIESSEN'; TextOff 'CLOSE / SCHLIESSEN'
      on Click: function_efd93a16("Template_Operating_Mode", 0, 0, 0, -1, 1)
      on Press: function_b14e0dd5("ButtonDown", 0)
      Appearance <- "ButtonDown"
   Button "Button_2" at 352,66 size 40x40; TextOff 'Text'; PictureOff "More_Icon"; PictureOn "More_Icon"
   Button "Button_3" at 352,130 size 40x40; TextOff 'Text'; PictureOff "More_Icon"; PictureOn "More_Icon"
   Button "Button_4" at 28,210 size 82x48; TextOff 'Start'
   Button "Button_5" at 123,210 size 82x48; TextOff 'Stop'
   Button "Button_6" at 218,210 size 82x48; TextOff 'Reset'
   Button "Button_7" at 314,210 size 82x48; TextOff 'Hold'
   TextField "txtParameter7_3" at 32,63 size 163x24; Text 'Current Mode'
   IOField "ioParameter17_3" at 32,81 size 301x40; FormatPattern ?????????????????????????
   TextField "txtParameter7_1" at 32,127 size 163x24; Text 'Current State'
   IOField "ioParameter17_1" at 32,145 size 301x40; FormatPattern ?????????????????????????

PopupScreen "Template_Recipe" 700x420
   on ClearScreen: ResetBit("PopUpBackground")
   on GenerateScreen: SetBit("PopUpBackground")
   TextField "Template_Text field_1" at 14,0 size 500x40; Text 'Recipe / Rezeptur'
   Button "Button_1" at 220,364 size 260x40; TextOn 'CLOSE / SCHLIESSEN'; TextOff 'CLOSE / SCHLIESSEN'
      on Click: function_efd93a16("Template_Recipe", 0, 0, 0, -1, 1)
      on Press: function_b14e0dd5("ButtonDown", 0)
      Appearance <- "ButtonDown"
   RecipeView "Rezepturanzeige_1" at 0,40 size 698x320

PopupScreen "OptionPanel_4_Buttons" 400x328
   GraphicView "gfxOptionPanel" at 80,30 size 18x12; Picture "ManFunctions_Off"
   TextField "textOptionPanelTitle" at 108,16 size 260x40; Text 'Option Panel Title / Titel Option Panel'
   Button "btnOptionPanelClose" at 0,0 size 40x328; TextOff 'Text'; PictureOff "Jog_Forward"
      on Press: function_efd93a16("OptionPanel_4_Buttons", 0, 0, 0, 2, 2)
   Button "btnOption1" at 80,72 size 240x40; TextOn 'Option 1'; TextOff 'Option 1 / Move to Home Position'
   Button "btnOption2" at 80,128 size 240x40; TextOn 'Option 2'; TextOff 'Option 2 / Move to Home Position'
   Button "btnOption3" at 80,184 size 240x40; TextOn 'Option 3'; TextOff 'Option 3 / RESET'
   Button "btnOption4" at 80,240 size 240x40; TextOn 'Option 4'; TextOff 'Option 4 / RESET'

SlideinScreen "GraphX_Slidein_Right" 220x480
   Button "Button_1" at 0,78 size 220x60; TextOn 'Menu Item 1'; TextOff 'Startscreen / Startseite'
      on Click: ActivateScreen("10_Startscreen", 0)
      Appearance <- "MainNavigationState"
   Button "Button_2" at 0,140 size 220x60; TextOn 'Menu Item 2'; TextOff 'Messages / Meldungen'
      on Click: ActivateScreen("20_Messages", 0)
      Appearance <- "MainNavigationState"
   Button "Button_3" at 0,201 size 220x60; TextOn 'Menu Item 3'; TextOff 'Diagnostics / Diagnose'
      on Click: ActivateScreen("30_Diagnostics", 0)
      Appearance <- "MainNavigationState"
   Rectangle "Rectangle_1" at 214,78 size 6x60
      Visibility <- "MainNavigationState"
   Rectangle "Rectangle_2" at 214,140 size 6x60
      Visibility <- "MainNavigationState"
   Rectangle "Rectangle_3" at 214,201 size 6x60
      Visibility <- "MainNavigationState"
   Button "Button_4" at 0,262 size 220x60; TextOn 'Menu Item 4'; TextOff 'Settings / Einstellungen'
      on Click: ActivateScreen("40_Settings", 0)
      Appearance <- "MainNavigationState"
   Rectangle "Rectangle_4" at 214,262 size 6x60
      Visibility <- "MainNavigationState"

VB script "ActivateAlarmControlScreen"
   bec8f1e5-2ab1-45f6-ad91-1d37c469eb91 20_Messages,0

VB script "ActivateStartScreen"
   HmiRuntime.BaseScreenName = SmartTags("StartScreenName")

VB script "CheckCurrentLanguage"
   If HmiRuntime.Language = 1031 Then 'German
   	SmartTags("CurrentLanguage") = 0
   	ElseIf HmiRuntime.Language = 1033 Then 'English US
   	SmartTags("CurrentLanguage") = 1
   End If
   
   	

VB script "CheckCurrentUserName"
   If SmartTags("CurrentUserName") = "" Or SmartTags("CurrentUserName") = "User Name" Or SmartTags("CurrentUserName") = "Benutzer" Then
     
     If HmiRuntime.Language = 1031 Then 'Germany
       SmartTags("CurrentUserName") = "Benutzer"
       
     ElseIf HmiRuntime.Language = 1033 Then 'English US
       SmartTags("CurrentUserName") = "User Name"
     End If
     
     SmartTags("UserIsLoggedIn") = False
   Else
     If SmartTags("CurrentUserName") <> "User Name" And SmartTags("CurrentUserName") <> "Benutzer" Then
       SmartTags("UserIsLoggedIn") = True  
     End If
   End If

VB script "CheckDiagState"
   If SmartTags("@DiagnosticsIndicatorTag") = 1 Then
   	SmartTags("DiagState") = 1
   Else
   	SmartTags("DiagState") = 0
   End If

VB script "GetStartScreenName"
   SmartTags("StartScreenName") = HmiRuntime.BaseScreenName

VB script "ShowLoginPopUp"
   efd93a16-2665-4b85-bcb9-25eddcb7b6f4 Template_Logon_Logoff,250,30,$3$hmiOn$,$3$hmiAnimationOff$,$3$hmiFast$

VB script "ShowOperatingModePopUp"
   efd93a16-2665-4b85-bcb9-25eddcb7b6f4 Template_Operating_Mode,188,30,$3$hmiOn$,$3$hmiAnimationOff$,$3$hmiFast$

VB script "ShowOptionPanelPopUp"
   efd93a16-2665-4b85-bcb9-25eddcb7b6f4 OptionPanel_4_Buttons, 410, 104, $3$hmiOn$, $3$hmiRight$, $3$hmiFast$

VB script "ShowRecipePopUp"
   efd93a16-2665-4b85-bcb9-25eddcb7b6f4 Template_Recipe,50,30,$3$hmiOn$,$3$hmiAnimationOff$,$3$hmiFast$

scheduled task "User Name"
   on Action: function_f41c6f6c("CurrentUserName"); "CheckCurrentUserName"()
*)